LIN {X 0,Y 566.191,Z 469.084,A -85,B 0,C 180,E1 -2638.953,E2 -2638.953} C_VEL
LIN {X 0,Y 566.2,Z 469.079,A -85,B 0,C 180,E1 -2641.421,E2 -2641.421} C_VEL
LIN {X 0,Y 566.208,Z 469.076,A -85,B 0,C 180,E1 -2643.955,E2 -2643.955} C_VEL
LIN {X 0,Y 566.197,Z 469.068,A -85,B 0,C 180,E1 -2646.569,E2 -2646.569} C_VEL
LIN {X 0,Y 566.219,Z 469.081,A -85,B 0,C 180,E1 -2649.272,E2 -2649.272} C_VEL
LIN {X 0,Y 566.211,Z 469.073,A -85,B 0,C 180,E1 -2652.086,E2 -2652.086} C_VEL
LIN {X 0,Y 566.169,Z 469.084,A -85,B 0,C 180,E1 -2655.035,E2 -2655.035} C_VEL
LIN {X 0,Y 566.186,Z 469.078,A -85,B 0,C 180,E1 -2657.91,E2 -2657.91} C_VEL
LIN {X 0,Y 566.217,Z 469.076,A -85,B 0,C 180,E1 -2660.726,E2 -2660.726} C_VEL
LIN {X 0,Y 566.212,Z 469.077,A -85,B 0,C 180,E1 -2663.783,E2 -2663.783} C_VEL
LIN {X 0,Y 566.206,Z 469.073,A -85,B 0,C 180,E1 -2666.265,E2 -2666.265} C_VEL
LIN {X 0,Y 566.192,Z 469.08,A -85,B 0,C 180,E1 -2668.921,E2 -2668.921} C_VEL
LIN {X 0,Y 566.221,Z 469.073,A -85,B 0,C 180,E1 -2671.858,E2 -2671.858} C_VEL
LIN {X 0,Y 566.219,Z 469.073,A -85,B 0,C 180,E1 -2674.251,E2 -2674.251} C_VEL
LIN {X 0,Y 566.183,Z 469.079,A -85,B 0,C 180,E1 -2676.713,E2 -2676.713} C_VEL
LIN {X 0,Y 566.211,Z 469.078,A -85,B 0,C 180,E1 -2679.662,E2 -2679.662} C_VEL
LIN {X 0,Y 566.195,Z 469.077,A -85,B 0,C 180,E1 -2682.668,E2 -2682.668} C_VEL
LIN {X 0,Y 566.224,Z 469.075,A -85,B 0,C 180,E1 -2685.626,E2 -2685.626} C_VEL
LIN {X 0,Y 566.224,Z 469.072,A -85,B 0,C 180,E1 -2688.675,E2 -2688.675} C_VEL
LIN {X 0,Y 566.24,Z 469.081,A -85,B 0,C 180,E1 -2691.434,E2 -2691.434} C_VEL
LIN {X 0,Y 566.252,Z 469.065,A -85,B 0,C 180,E1 -2694.301,E2 -2694.301} C_VEL
LIN {X 0,Y 566.272,Z 469.071,A -85,B 0,C 180,E1 -2697.866,E2 -2697.866} C_VEL
LIN {X 0,Y 566.298,Z 469.062,A -85,B 0,C 180,E1 -2700.711,E2 -2700.711} C_VEL
LIN {X 0,Y 566.27,Z 469.064,A -85,B 0,C 180,E1 -2702.845,E2 -2702.845} C_VEL
LIN {X 0,Y 566.25,Z 469.077,A -85,B 0,C 180,E1 -2705.698,E2 -2705.698} C_VEL
LIN {X 0,Y 566.239,Z 469.069,A -85,B 0,C 180,E1 -2708.565,E2 -2708.565} C_VEL
LIN {X 0,Y 566.241,Z 469.076,A -85,B 0,C 180,E1 -2711.454,E2 -2711.454} C_VEL
LIN {X 0,Y 566.223,Z 469.073,A -85,B 0,C 180,E1 -2714.507,E2 -2714.507} C_VEL
LIN {X 0,Y 566.194,Z 469.08,A -85,B 0,C 180,E1 -2717.331,E2 -2717.331} C_VEL
LIN {X 0,Y 566.21,Z 469.075,A -85,B 0,C 180,E1 -2720.337,E2 -2720.337} C_VEL
LIN {X 0,Y 566.179,Z 469.084,A -85,B 0,C 180,E1 -2723.404,E2 -2723.404} C_VEL
LIN {X 0,Y 566.217,Z 469.082,A -85,B 0,C 180,E1 -2725.748,E2 -2725.748} C_VEL
LIN {X 0,Y 566.207,Z 469.078,A -85,B 0,C 180,E1 -2727.497,E2 -2727.497} C_VEL
LIN {X 0,Y 565.529,Z 469.163,A -85,B 0,C 180,E1 -2728.09,E2 -2728.09} C_VEL
LIN {X 0,Y 562.664,Z 469.517,A -85,B 0,C 180,E1 -2729.054,E2 -2729.054} C_VEL
LIN {X 0,Y 560.253,Z 469.821,A -85,B 0,C 180,E1 -2729.83,E2 -2729.83} C_VEL
LIN {X 0,Y 559.224,Z 469.943,A -85,B 0,C 180,E1 -2730.428,E2 -2730.428} C_VEL
LIN {X 0,Y 559.143,Z 469.952,A -85,B 0,C 180,E1 -2730.631,E2 -2730.631} C_VEL
LIN {X 0,Y 559.169,Z 469.96,A -85,B 0,C 180,E1 -2733.574,E2 -2733.574} C_VEL
LIN {X 0,Y 559.16,Z 469.952,A -85,B 0,C 180,E1 -2736.449,E2 -2736.449} C_VEL
LIN {X 0,Y 559.17,Z 469.952,A -85,B 0,C 180,E1 -2738.934,E2 -2738.934} C_VEL
LIN {X 0,Y 559.183,Z 469.959,A -85,B 0,C 180,E1 -2741.768,E2 -2741.768} C_VEL
LIN {X 0,Y 559.131,Z 469.955,A -85,B 0,C 180,E1 -2744.739,E2 -2744.739} C_VEL
LIN {X 0,Y 559.165,Z 469.946,A -85,B 0,C 180,E1 -2747.258,E2 -2747.258} C_VEL
LIN {X 0,Y 559.179,Z 469.955,A -85,B 0,C 180,E1 -2750.135,E2 -2750.135} C_VEL
LIN {X 0,Y 559.14,Z 469.951,A -85,B 0,C 180,E1 -2752.893,E2 -2752.893} C_VEL
LIN {X 0,Y 559.149,Z 469.96,A -85,B 0,C 180,E1 -2755.556,E2 -2755.556} C_VEL
LIN {X 0,Y 559.165,Z 469.958,A -85,B 0,C 180,E1 -2758.138,E2 -2758.138} C_VEL
LIN {X 0,Y 559.151,Z 469.955,A -85,B 0,C 180,E1 -2760.647,E2 -2760.647} C_VEL
LIN {X 0,Y 559.166,Z 469.954,A -85,B 0,C 180,E1 -2763.173,E2 -2763.173} C_VEL
LIN {X 0,Y 559.152,Z 469.959,A -85,B 0,C 180,E1 -2765.495,E2 -2765.495} C_VEL
LIN {X 0,Y 559.167,Z 469.954,A -85,B 0,C 180,E1 -2768.624,E2 -2768.624} C_VEL
LIN {X 0,Y 559.166,Z 469.953,A -85,B 0,C 180,E1 -2770.927,E2 -2770.927} C_VEL
LIN {X 0,Y 559.164,Z 469.962,A -85,B 0,C 180,E1 -2773.948,E2 -2773.948} C_VEL
LIN {X 0,Y 559.169,Z 469.959,A -85,B 0,C 180,E1 -2776.184,E2 -2776.184} C_VEL
LIN {X 0,Y 559.191,Z 469.951,A -85,B 0,C 180,E1 -2779.134,E2 -2779.134} C_VEL
LIN {X 0,Y 559.202,Z 469.957,A -85,B 0,C 180,E1 -2782.054,E2 -2782.054} C_VEL
LIN {X 0,Y 559.248,Z 469.943,A -85,B 0,C 180,E1 -2784.953,E2 -2784.953} C_VEL
LIN {X 0,Y 559.252,Z 469.951,A -85,B 0,C 180,E1 -2787.839,E2 -2787.839} C_VEL
LIN {X 0,Y 559.268,Z 469.942,A -85,B 0,C 180,E1 -2790.72,E2 -2790.72} C_VEL
LIN {X 0,Y 559.235,Z 469.945,A -85,B 0,C 180,E1 -2792.881,E2 -2792.881} C_VEL
LIN {X 0,Y 559.225,Z 469.952,A -85,B 0,C 180,E1 -2795.77,E2 -2795.77} C_VEL
LIN {X 0,Y 559.183,Z 469.952,A -85,B 0,C 180,E1 -2798.674,E2 -2798.674} C_VEL
LIN {X 0,Y 559.202,Z 469.952,A -85,B 0,C 180,E1 -2801.6,E2 -2801.6} C_VEL
LIN {X 0,Y 559.196,Z 469.952,A -85,B 0,C 180,E1 -2804.595,E2 -2804.595} C_VEL
LIN {X 0,Y 559.159,Z 469.956,A -85,B 0,C 180,E1 -2807.556,E2 -2807.556} C_VEL
LIN {X 0,Y 559.168,Z 469.959,A -85,B 0,C 180,E1 -2809.837,E2 -2809.837} C_VEL
LIN {X 0,Y 559.137,Z 469.966,A -85,B 0,C 180,E1 -2812.152,E2 -2812.152} C_VEL
LIN {X 0,Y 559.174,Z 469.952,A -85,B 0,C 180,E1 -2815.187,E2 -2815.187} C_VEL
LIN {X 0,Y 559.186,Z 469.954,A -85,B 0,C 180,E1 -2817.711,E2 -2817.711} C_VEL
LIN {X 0,Y 559.163,Z 469.963,A -85,B 0,C 180,E1 -2820.181,E2 -2820.181} C_VEL
LIN {X 0,Y 559.169,Z 469.955,A -85,B 0,C 180,E1 -2822.714,E2 -2822.714} C_VEL
LIN {X 0,Y 559.15,Z 469.954,A -85,B 0,C 180,E1 -2825.322,E2 -2825.322} C_VEL
LIN {X 0,Y 559.129,Z 469.96,A -85,B 0,C 180,E1 -2828.017,E2 -2828.017} C_VEL
LIN {X 0,Y 559.169,Z 469.952,A -85,B 0,C 180,E1 -2830.81,E2 -2830.81} C_VEL
LIN {X 0,Y 559.156,Z 469.947,A -85,B 0,C 180,E1 -2833.731,E2 -2833.731} C_VEL
LIN {X 0,Y 559.159,Z 469.956,A -85,B 0,C 180,E1 -2836.801,E2 -2836.801} C_VEL
LIN {X 0,Y 559.167,Z 469.95,A -85,B 0,C 180,E1 -2839.189,E2 -2839.189} C_VEL
LIN {X 0,Y 559.126,Z 469.963,A -85,B 0,C 180,E1 -2841.982,E2 -2841.982} C_VEL
LIN {X 0,Y 559.152,Z 469.956,A -85,B 0,C 180,E1 -2844.782,E2 -2844.782} C_VEL
LIN {X 0,Y 559.165,Z 469.952,A -85,B 0,C 180,E1 -2847.361,E2 -2847.361} C_VEL
LIN {X 0,Y 559.18,Z 469.954,A -85,B 0,C 180,E1 -2850.135,E2 -2850.135} C_VEL
LIN {X 0,Y 559.173,Z 469.951,A -85,B 0,C 180,E1 -2853.17,E2 -2853.17} C_VEL
LIN {X 0,Y 559.147,Z 469.951,A -85,B 0,C 180,E1 -2855.495,E2 -2855.495} C_VEL
LIN {X 0,Y 559.167,Z 469.958,A -85,B 0,C 180,E1 -2858.624,E2 -2858.624} C_VEL
LIN {X 0,Y 559.162,Z 469.953,A -85,B 0,C 180,E1 -2860.926,E2 -2860.926} C_VEL
LIN {X 0,Y 559.161,Z 469.953,A -85,B 0,C 180,E1 -2863.948,E2 -2863.948} C_VEL
LIN {X 0,Y 559.164,Z 469.958,A -85,B 0,C 180,E1 -2866.184,E2 -2866.184} C_VEL
LIN {X 0,Y 559.201,Z 469.945,A -85,B 0,C 180,E1 -2869.134,E2 -2869.134} C_VEL
LIN {X 0,Y 559.201,Z 469.949,A -85,B 0,C 180,E1 -2872.054,E2 -2872.054} C_VEL
LIN {X 0,Y 559.251,Z 469.943,A -85,B 0,C 180,E1 -2874.954,E2 -2874.954} C_VEL
LIN {X 0,Y 559.243,Z 469.939,A -85,B 0,C 180,E1 -2877.84,E2 -2877.84} C_VEL
LIN {X 0,Y 559.268,Z 469.945,A -85,B 0,C 180,E1 -2880.72,E2 -2880.72} C_VEL
LIN {X 0,Y 559.236,Z 469.946,A -85,B 0,C 180,E1 -2882.882,E2 -2882.882} C_VEL
LIN {X 0,Y 559.221,Z 469.94,A -85,B 0,C 180,E1 -2885.771,E2 -2885.771} C_VEL
LIN {X 0,Y 559.194,Z 469.957,A -85,B 0,C 180,E1 -2888.675,E2 -2888.675} C_VEL
LIN {X 0,Y 559.196,Z 469.947,A -85,B 0,C 180,E1 -2891.601,E2 -2891.601} C_VEL
LIN {X 0,Y 559.19,Z 469.955,A -85,B 0,C 180,E1 -2894.596,E2 -2894.596} C_VEL
LIN {X 0,Y 559.155,Z 469.953,A -85,B 0,C 180,E1 -2897.557,E2 -2897.557} C_VEL
LIN {X 0,Y 559.166,Z 469.95,A -85,B 0,C 180,E1 -2899.838,E2 -2899.838} C_VEL
LIN {X 0,Y 559.135,Z 469.957,A -85,B 0,C 180,E1 -2902.153,E2 -2902.153} C_VEL
LIN {X 0,Y 559.172,Z 469.952,A -85,B 0,C 180,E1 -2905.188,E2 -2905.188} C_VEL
LIN {X 0,Y 559.188,Z 469.946,A -85,B 0,C 180,E1 -2907.712,E2 -2907.712} C_VEL
LIN {X 0,Y 559.156,Z 469.957,A -85,B 0,C 180,E1 -2911.02,E2 -2911.02} C_VEL
LIN {X 0,Y 559.162,Z 469.951,A -85,B 0,C 180,E1 -2913.95,E2 -2913.95} C_VEL
LIN {X 0,Y 559.163,Z 469.959,A -85,B 0,C 180,E1 -2916.449,E2 -2916.449} C_VEL
LIN {X 0,Y 559.173,Z 469.958,A -85,B 0,C 180,E1 -2918.934,E2 -2918.934} C_VEL
LIN {X 0,Y 559.164,Z 469.951,A -85,B 0,C 180,E1 -2921.77,E2 -2921.77} C_VEL
LIN {X 0,Y 559.135,Z 469.965,A -85,B 0,C 180,E1 -2924.74,E2 -2924.74} C_VEL
LIN {X 0,Y 559.161,Z 469.954,A -85,B 0,C 180,E1 -2927.258,E2 -2927.258} C_VEL
LIN {X 0,Y 559.182,Z 469.952,A -85,B 0,C 180,E1 -2930.136,E2 -2930.136} C_VEL
LIN {X 0,Y 559.138,Z 469.95,A -85,B 0,C 180,E1 -2932.892,E2 -2932.892} C_VEL
LIN {X 0,Y 559.164,Z 469.954,A -85,B 0,C 180,E1 -2936.052,E2 -2936.052} C_VEL
LIN {X 0,Y 559.162,Z 469.951,A -85,B 0,C 180,E1 -2938.982,E2 -2938.982} C_VEL
LIN {X 0,Y 559.168,Z 469.953,A -85,B 0,C 180,E1 -2941.619,E2 -2941.619} C_VEL
LIN {X 0,Y 559.2,Z 470.086,A -85,B 0,C 180,E1 -2943.503,E2 -2943.503} C_VEL
LIN {X 0,Y 560.282,Z 475.94,A -85,B 0,C 180,E1 -2944.575,E2 -2944.575} C_VEL
LIN {X 0,Y 560.031,Z 493.496,A -85,B 0,C 180,E1 -2947.496,E2 -2947.496} C_VEL
LIN {X 0,Y 559.744,Z 510.701,A -85,B 0,C 180,E1 -2950.336,E2 -2950.336} C_VEL
LIN {X 0,Y 559.551,Z 526.039,A -85,B 0,C 180,E1 -2952.795,E2 -2952.795} C_VEL
LIN {X 0,Y 560.706,Z 532.012,A -85,B 0,C 180,E1 -2952.937,E2 -2952.937} C_VEL
LIN {X 0,Y 561.014,Z 537.106,A -85,B 0,C 180,E1 -2953.014,E2 -2953.014} C_VEL
LIN {X 0,Y 560.621,Z 661.281,A -85,B 0,C 180,E1 -2954.644,E2 -2954.644} C_VEL
LIN {X 0,Y 560.468,Z 673.415,A -85,B 0,C 180,E1 -2954.905,E2 -2954.905} C_VEL
LIN {X 0,Y 560.366,Z 685.467,A -85,B 0,C 180,E1 -2955.275,E2 -2955.275} C_VEL
LIN {X 0,Y 560.152,Z 699.181,A -85,B 0,C 180,E1 -2955.839,E2 -2955.839} C_VEL
LIN {X 0,Y 559.865,Z 712.711,A -85,B 0,C 180,E1 -2956.572,E2 -2956.572} C_VEL
LIN {X 0,Y 559.702,Z 723.64,A -85,B 0,C 180,E1 -2957.306,E2 -2957.306} C_VEL
LIN {X 0,Y 559.514,Z 733.886,A -85,B 0,C 180,E1 -2958.131,E2 -2958.131} C_VEL
LIN {X 0,Y 559.35,Z 744.375,A -85,B 0,C 180,E1 -2959.137,E2 -2959.137} C_VEL
LIN {X 0,Y 559.143,Z 753.825,A -85,B 0,C 180,E1 -2960.231,E2 -2960.231} C_VEL
LIN {X 0,Y 559.053,Z 761.624,A -85,B 0,C 180,E1 -2961.324,E2 -2961.324} C_VEL
LIN {X 0,Y 558.966,Z 768.13,A -85,B 0,C 180,E1 -2962.414,E2 -2962.414} C_VEL
LIN {X 0,Y 558.872,Z 773.519,A -85,B 0,C 180,E1 -2963.502,E2 -2963.502} C_VEL
LIN {X 0,Y 558.858,Z 777.921,A -85,B 0,C 180,E1 -2964.588,E2 -2964.588} C_VEL
LIN {X 0,Y 558.865,Z 781.441,A -85,B 0,C 180,E1 -2965.673,E2 -2965.673} C_VEL
LIN {X 0,Y 558.825,Z 783.323,A -85,B 0,C 180,E1 -2966.395,E2 -2966.395} C_VEL
LIN {X 0,Y 558.743,Z 786.005,A -85,B 0,C 180,E1 -2967.837,E2 -2967.837} C_VEL
LIN {X 0,Y 558.738,Z 787.29,A -85,B 0,C 180,E1 -2969.279,E2 -2969.279} C_VEL
LIN {X 0,Y 558.738,Z 787.5,A -85,B 0,C 180,E1 -2970,E2 -2970} C_VEL
LIN {X 0,Y 558.74,Z 786.808,A -85,B 0,C 180,E1 -2971.441,E2 -2971.441} C_VEL
LIN {X 0,Y 558.743,Z 786.005,A -85,B 0,C 180,E1 -2972.163,E2 -2972.163} C_VEL
LIN {X 0,Y 558.825,Z 783.323,A -85,B 0,C 180,E1 -2973.605,E2 -2973.605} C_VEL
LIN {X 0,Y 558.82,Z 780.397,A -85,B 0,C 180,E1 -2974.689,E2 -2974.689} C_VEL
LIN {X 0,Y 558.882,Z 775.086,A -85,B 0,C 180,E1 -2976.136,E2 -2976.136} C_VEL
LIN {X 0,Y 558.907,Z 770.03,A -85,B 0,C 180,E1 -2977.224,E2 -2977.224} C_VEL
LIN {X 0,Y 559.006,Z 763.885,A -85,B 0,C 180,E1 -2978.313,E2 -2978.313} C_VEL
LIN {X 0,Y 559.117,Z 756.524,A -85,B 0,C 180,E1 -2979.405,E2 -2979.405} C_VEL
LIN {X 0,Y 559.267,Z 747.714,A -85,B 0,C 180,E1 -2980.498,E2 -2980.498} C_VEL
LIN {X 0,Y 559.454,Z 737.023,A -85,B 0,C 180,E1 -2981.595,E2 -2981.595} C_VEL
LIN {X 0,Y 559.637,Z 726.113,A -85,B 0,C 180,E1 -2982.511,E2 -2982.511} C_VEL
LIN {X 0,Y 559.827,Z 715.633,A -85,B 0,C 180,E1 -2983.244,E2 -2983.244} C_VEL
LIN {X 0,Y 560.047,Z 704.551,A -85,B 0,C 180,E1 -2983.886,E2 -2983.886} C_VEL
LIN {X 0,Y 560.232,Z 692.882,A -85,B 0,C 180,E1 -2984.437,E2 -2984.437} C_VEL
LIN {X 0,Y 560.411,Z 679.335,A -85,B 0,C 180,E1 -2984.933,E2 -2984.933} C_VEL
LIN {X 0,Y 560.563,Z 663.998,A -85,B 0,C 180,E1 -2985.311,E2 -2985.311} C_VEL
LIN {X 0,Y 560.693,Z 637.754,A -85,B 0,C 180,E1 -2985.68,E2 -2985.68} C_VEL
LIN {X 0,Y 560.863,Z 532.996,A -85,B 0,C 180,E1 -2987.045,E2 -2987.045} C_VEL
LIN {X 0,Y 559.547,Z 526.183,A -85,B 0,C 180,E1 -2987.195,E2 -2987.195} C_VEL
LIN {X 0,Y 559.567,Z 522.568,A -85,B 0,C 180,E1 -2987.732,E2 -2987.732} C_VEL
LIN {X 0,Y 559.837,Z 503.962,A -85,B 0,C 180,E1 -2990.771,E2 -2990.771} C_VEL
LIN {X 0,Y 560.096,Z 488.81,A -85,B 0,C 180,E1 -2993.281,E2 -2993.281} C_VEL
LIN {X 0,Y 560.269,Z 475.96,A -85,B 0,C 180,E1 -2995.422,E2 -2995.422} C_VEL
LIN {X 0,Y 559.19,Z 470.039,A -85,B 0,C 180,E1 -2996.518,E2 -2996.518} C_VEL
LIN {X 0,Y 559.142,Z 469.962,A -85,B 0,C 180,E1 -2999.353,E2 -2999.353} C_VEL
LIN {X 0,Y 559.169,Z 469.952,A -85,B 0,C 180,E1 -3001.862,E2 -3001.862} C_VEL
LIN {X 0,Y 559.141,Z 469.957,A -85,B 0,C 180,E1 -3004.444,E2 -3004.444} C_VEL
LIN {X 0,Y 559.138,Z 469.95,A -85,B 0,C 180,E1 -3007.108,E2 -3007.108} C_VEL
LIN {X 0,Y 559.166,Z 469.953,A -85,B 0,C 180,E1 -3009.942,E2 -3009.942} C_VEL
LIN {X 0,Y 559.161,Z 469.954,A -85,B 0,C 180,E1 -3012.742,E2 -3012.742} C_VEL
LIN {X 0,Y 559.148,Z 469.957,A -85,B 0,C 180,E1 -3015.76,E2 -3015.76} C_VEL
LIN {X 0,Y 559.164,Z 469.951,A -85,B 0,C 180,E1 -3018.23,E2 -3018.23} C_VEL
LIN {X 0,Y 559.172,Z 469.96,A -85,B 0,C 180,E1 -3021.19,E2 -3021.19} C_VEL
LIN {X 0,Y 559.167,Z 469.955,A -85,B 0,C 180,E1 -3023.791,E2 -3023.791} C_VEL
LIN {X 0,Y 559.159,Z 469.951,A -85,B 0,C 180,E1 -3026.425,E2 -3026.425} C_VEL
LIN {X 0,Y 559.156,Z 469.957,A -85,B 0,C 180,E1 -3028.98,E2 -3028.98} C_VEL
LIN {X 0,Y 559.188,Z 469.946,A -85,B 0,C 180,E1 -3032.288,E2 -3032.288} C_VEL
LIN {X 0,Y 559.172,Z 469.952,A -85,B 0,C 180,E1 -3034.812,E2 -3034.812} C_VEL
LIN {X 0,Y 559.135,Z 469.957,A -85,B 0,C 180,E1 -3037.847,E2 -3037.847} C_VEL
LIN {X 0,Y 559.19,Z 469.947,A -85,B 0,C 180,E1 -3040.491,E2 -3040.491} C_VEL
LIN {X 0,Y 559.176,Z 469.957,A -85,B 0,C 180,E1 -3043.197,E2 -3043.197} C_VEL
LIN {X 0,Y 559.164,Z 469.948,A -85,B 0,C 180,E1 -3046.184,E2 -3046.184} C_VEL
LIN {X 0,Y 559.187,Z 469.953,A -85,B 0,C 180,E1 -3049.133,E2 -3049.133} C_VEL
LIN {X 0,Y 559.2,Z 469.948,A -85,B 0,C 180,E1 -3052.053,E2 -3052.053} C_VEL
LIN {X 0,Y 559.25,Z 469.939,A -85,B 0,C 180,E1 -3054.953,E2 -3054.953} C_VEL
LIN {X 0,Y 559.243,Z 469.947,A -85,B 0,C 180,E1 -3057.839,E2 -3057.839} C_VEL
LIN {X 0,Y 559.268,Z 469.937,A -85,B 0,C 180,E1 -3060.72,E2 -3060.72} C_VEL
LIN {X 0,Y 559.236,Z 469.94,A -85,B 0,C 180,E1 -3062.881,E2 -3062.881} C_VEL
LIN {X 0,Y 559.22,Z 469.951,A -85,B 0,C 180,E1 -3065.77,E2 -3065.77} C_VEL
LIN {X 0,Y 559.194,Z 469.946,A -85,B 0,C 180,E1 -3068.674,E2 -3068.674} C_VEL
LIN {X 0,Y 559.199,Z 469.955,A -85,B 0,C 180,E1 -3071.6,E2 -3071.6} C_VEL
LIN {X 0,Y 559.188,Z 469.949,A -85,B 0,C 180,E1 -3074.595,E2 -3074.595} C_VEL
LIN {X 0,Y 559.154,Z 469.959,A -85,B 0,C 180,E1 -3077.557,E2 -3077.557} C_VEL
LIN {X 0,Y 559.165,Z 469.959,A -85,B 0,C 180,E1 -3079.837,E2 -3079.837} C_VEL
LIN {X 0,Y 559.132,Z 469.958,A -85,B 0,C 180,E1 -3082.153,E2 -3082.153} C_VEL
LIN {X 0,Y 559.169,Z 469.951,A -85,B 0,C 180,E1 -3085.187,E2 -3085.187} C_VEL
LIN {X 0,Y 559.185,Z 469.959,A -85,B 0,C 180,E1 -3087.711,E2 -3087.711} C_VEL
LIN {X 0,Y 559.143,Z 469.952,A -85,B 0,C 180,E1 -3090.631,E2 -3090.631} C_VEL
LIN {X 0,Y 558.48,Z 470.039,A -85,B 0,C 180,E1 -3091.233,E2 -3091.233} C_VEL
LIN {X 0,Y 555.617,Z 470.396,A -85,B 0,C 180,E1 -3092.209,E2 -3092.209} C_VEL
LIN {X 0,Y 553.206,Z 470.696,A -85,B 0,C 180,E1 -3092.994,E2 -3092.994} C_VEL
LIN {X 0,Y 552.188,Z 470.83,A -85,B 0,C 180,E1 -3093.601,E2 -3093.601} C_VEL
LIN {X 0,Y 552.115,Z 470.832,A -85,B 0,C 180,E1 -3093.806,E2 -3093.806} C_VEL
LIN {X 0,Y 552.103,Z 470.83,A -85,B 0,C 180,E1 -3096.747,E2 -3096.747} C_VEL
LIN {X 0,Y 552.126,Z 470.836,A -85,B 0,C 180,E1 -3099.527,E2 -3099.527} C_VEL
LIN {X 0,Y 552.122,Z 470.831,A -85,B 0,C 180,E1 -3102.426,E2 -3102.426} C_VEL
LIN {X 0,Y 552.092,Z 470.839,A -85,B 0,C 180,E1 -3105.563,E2 -3105.563} C_VEL
LIN {X 0,Y 552.164,Z 470.823,A -85,B 0,C 180,E1 -3108.673,E2 -3108.673} C_VEL
LIN {X 0,Y 552.114,Z 470.835,A -85,B 0,C 180,E1 -3111.412,E2 -3111.412} C_VEL
LIN {X 0,Y 552.106,Z 470.836,A -85,B 0,C 180,E1 -3114.159,E2 -3114.159} C_VEL
LIN {X 0,Y 552.117,Z 470.831,A -85,B 0,C 180,E1 -3116.815,E2 -3116.815} C_VEL
LIN {X 0,Y 552.108,Z 470.835,A -85,B 0,C 180,E1 -3119.392,E2 -3119.392} C_VEL
LIN {X 0,Y 552.12,Z 470.84,A -85,B 0,C 180,E1 -3121.903,E2 -3121.903} C_VEL
LIN {X 0,Y 552.15,Z 470.828,A -85,B 0,C 180,E1 -3124.65,E2 -3124.65} C_VEL
LIN {X 0,Y 552.091,Z 470.839,A -85,B 0,C 180,E1 -3127.55,E2 -3127.55} C_VEL
LIN {X 0,Y 552.152,Z 470.828,A -85,B 0,C 180,E1 -3130.675,E2 -3130.675} C_VEL
LIN {X 0,Y 552.114,Z 470.839,A -85,B 0,C 180,E1 -3133.738,E2 -3133.738} C_VEL
LIN {X 0,Y 552.132,Z 470.838,A -85,B 0,C 180,E1 -3136.005,E2 -3136.005} C_VEL
LIN {X 0,Y 552.159,Z 470.826,A -85,B 0,C 180,E1 -3138.994,E2 -3138.994} C_VEL
LIN {X 0,Y 552.156,Z 470.835,A -85,B 0,C 180,E1 -3141.952,E2 -3141.952} C_VEL
LIN {X 0,Y 552.223,Z 470.819,A -85,B 0,C 180,E1 -3144.889,E2 -3144.889} C_VEL
LIN {X 0,Y 552.223,Z 470.826,A -85,B 0,C 180,E1 -3147.812,E2 -3147.812} C_VEL
LIN {X 0,Y 552.238,Z 470.818,A -85,B 0,C 180,E1 -3150.729,E2 -3150.729} C_VEL
LIN {X 0,Y 552.202,Z 470.821,A -85,B 0,C 180,E1 -3152.918,E2 -3152.918} C_VEL
LIN {X 0,Y 552.196,Z 470.829,A -85,B 0,C 180,E1 -3155.844,E2 -3155.844} C_VEL
LIN {X 0,Y 552.154,Z 470.827,A -85,B 0,C 180,E1 -3158.786,E2 -3158.786} C_VEL
LIN {X 0,Y 552.159,Z 470.831,A -85,B 0,C 180,E1 -3161.75,E2 -3161.75} C_VEL
LIN {X 0,Y 552.133,Z 470.831,A -85,B 0,C 180,E1 -3164.748,E2 -3164.748} C_VEL
LIN {X 0,Y 552.11,Z 470.838,A -85,B 0,C 180,E1 -3167.788,E2 -3167.788} C_VEL
LIN {X 0,Y 552.126,Z 470.839,A -85,B 0,C 180,E1 -3170.101,E2 -3170.101} C_VEL
LIN {X 0,Y 552.091,Z 470.839,A -85,B 0,C 180,E1 -3172.45,E2 -3172.45} C_VEL
LIN {X 0,Y 552.15,Z 470.828,A -85,B 0,C 180,E1 -3175.35,E2 -3175.35} C_VEL
LIN {X 0,Y 552.12,Z 470.84,A -85,B 0,C 180,E1 -3178.097,E2 -3178.097} C_VEL
LIN {X 0,Y 552.108,Z 470.835,A -85,B 0,C 180,E1 -3180.608,E2 -3180.608} C_VEL
LIN {X 0,Y 552.117,Z 470.831,A -85,B 0,C 180,E1 -3183.185,E2 -3183.185} C_VEL
LIN {X 0,Y 552.106,Z 470.836,A -85,B 0,C 180,E1 -3185.841,E2 -3185.841} C_VEL
LIN {X 0,Y 552.119,Z 470.831,A -85,B 0,C 180,E1 -3189.062,E2 -3189.062} C_VEL
LIN {X 0,Y 552.134,Z 470.827,A -85,B 0,C 180,E1 -3191.443,E2 -3191.443} C_VEL
LIN {X 0,Y 552.089,Z 470.838,A -85,B 0,C 180,E1 -3194.532,E2 -3194.532} C_VEL
LIN {X 0,Y 552.122,Z 470.831,A -85,B 0,C 180,E1 -3197.584,E2 -3197.584} C_VEL
LIN {X 0,Y 552.126,Z 470.836,A -85,B 0,C 180,E1 -3200.473,E2 -3200.473} C_VEL
LIN {X 0,Y 552.105,Z 470.83,A -85,B 0,C 180,E1 -3203.315,E2 -3203.315} C_VEL
LIN {X 0,Y 552.131,Z 470.832,A -85,B 0,C 180,E1 -3205.94,E2 -3205.94} C_VEL
LIN {X 0,Y 552.108,Z 470.834,A -85,B 0,C 180,E1 -3208.54,E2 -3208.54} C_VEL
LIN {X 0,Y 552.117,Z 470.83,A -85,B 0,C 180,E1 -3211.437,E2 -3211.437} C_VEL
LIN {X 0,Y 552.128,Z 470.835,A -85,B 0,C 180,E1 -3214.356,E2 -3214.356} C_VEL
LIN {X 0,Y 552.1,Z 470.835,A -85,B 0,C 180,E1 -3216.758,E2 -3216.758} C_VEL
LIN {X 0,Y 552.116,Z 470.831,A -85,B 0,C 180,E1 -3219.12,E2 -3219.12} C_VEL
LIN {X 0,Y 552.122,Z 470.827,A -85,B 0,C 180,E1 -3221.445,E2 -3221.445} C_VEL
LIN {X 0,Y 552.111,Z 470.829,A -85,B 0,C 180,E1 -3223.738,E2 -3223.738} C_VEL
LIN {X 0,Y 552.126,Z 470.832,A -85,B 0,C 180,E1 -3226.005,E2 -3226.005} C_VEL
LIN {X 0,Y 552.168,Z 470.822,A -85,B 0,C 180,E1 -3228.994,E2 -3228.994} C_VEL
LIN {X 0,Y 552.155,Z 470.825,A -85,B 0,C 180,E1 -3231.952,E2 -3231.952} C_VEL
LIN {X 0,Y 552.225,Z 470.819,A -85,B 0,C 180,E1 -3234.889,E2 -3234.889} C_VEL
LIN {X 0,Y 552.215,Z 470.814,A -85,B 0,C 180,E1 -3237.812,E2 -3237.812} C_VEL
LIN {X 0,Y 552.237,Z 470.821,A -85,B 0,C 180,E1 -3240.73,E2 -3240.73} C_VEL
LIN {X 0,Y 552.202,Z 470.822,A -85,B 0,C 180,E1 -3242.918,E2 -3242.918} C_VEL
LIN {X 0,Y 552.191,Z 470.816,A -85,B 0,C 180,E1 -3245.844,E2 -3245.844} C_VEL
LIN {X 0,Y 552.162,Z 470.831,A -85,B 0,C 180,E1 -3248.786,E2 -3248.786} C_VEL
LIN {X 0,Y 552.153,Z 470.825,A -85,B 0,C 180,E1 -3251.751,E2 -3251.751} C_VEL
LIN {X 0,Y 552.128,Z 470.835,A -85,B 0,C 180,E1 -3254.749,E2 -3254.749} C_VEL
LIN {X 0,Y 552.107,Z 470.832,A -85,B 0,C 180,E1 -3257.789,E2 -3257.789} C_VEL
LIN {X 0,Y 552.126,Z 470.829,A -85,B 0,C 180,E1 -3260.102,E2 -3260.102} C_VEL
LIN {X 0,Y 552.088,Z 470.838,A -85,B 0,C 180,E1 -3262.451,E2 -3262.451} C_VEL
LIN {X 0,Y 552.149,Z 470.826,A -85,B 0,C 180,E1 -3265.352,E2 -3265.352} C_VEL
LIN {X 0,Y 552.12,Z 470.829,A -85,B 0,C 180,E1 -3268.098,E2 -3268.098} C_VEL
LIN {X 0,Y 552.101,Z 470.842,A -85,B 0,C 180,E1 -3270.61,E2 -3270.61} C_VEL
LIN {X 0,Y 552.117,Z 470.831,A -85,B 0,C 180,E1 -3273.186,E2 -3273.186} C_VEL
LIN {X 0,Y 552.108,Z 470.832,A -85,B 0,C 180,E1 -3275.842,E2 -3275.842} C_VEL
LIN {X 0,Y 552.12,Z 470.835,A -85,B 0,C 180,E1 -3279.063,E2 -3279.063} C_VEL
LIN {X 0,Y 552.125,Z 470.829,A -85,B 0,C 180,E1 -3281.446,E2 -3281.446} C_VEL
LIN {X 0,Y 552.091,Z 470.841,A -85,B 0,C 180,E1 -3284.533,E2 -3284.533} C_VEL
LIN {X 0,Y 552.128,Z 470.827,A -85,B 0,C 180,E1 -3287.585,E2 -3287.585} C_VEL
LIN {X 0,Y 552.131,Z 470.834,A -85,B 0,C 180,E1 -3290.474,E2 -3290.474} C_VEL
LIN {X 0,Y 552.104,Z 470.821,A -85,B 0,C 180,E1 -3293.318,E2 -3293.318} C_VEL
LIN {X 0,Y 552.125,Z 470.831,A -85,B 0,C 180,E1 -3295.94,E2 -3295.94} C_VEL
LIN {X 0,Y 552.118,Z 470.831,A -85,B 0,C 180,E1 -3298.541,E2 -3298.541} C_VEL
LIN {X 0,Y 552.124,Z 470.831,A -85,B 0,C 180,E1 -3301.439,E2 -3301.439} C_VEL
LIN {X 0,Y 552.17,Z 471.047,A -85,B 0,C 180,E1 -3303.339,E2 -3303.339} C_VEL
LIN {X 0,Y 553.38,Z 477.467,A -85,B 0,C 180,E1 -3304.524,E2 -3304.524} C_VEL
LIN {X 0,Y 553.086,Z 495.719,A -85,B 0,C 180,E1 -3307.592,E2 -3307.592} C_VEL
LIN {X 0,Y 552.742,Z 512.913,A -85,B 0,C 180,E1 -3310.445,E2 -3310.445} C_VEL
LIN {X 0,Y 552.607,Z 526.043,A -85,B 0,C 180,E1 -3312.572,E2 -3312.572} C_VEL
LIN {X 0,Y 553.554,Z 531.047,A -85,B 0,C 180,E1 -3312.697,E2 -3312.697} C_VEL
LIN {X 0,Y 554.245,Z 535.775,A -85,B 0,C 180,E1 -3312.782,E2 -3312.782} C_VEL
LIN {X 0,Y 553.785,Z 661.233,A -85,B 0,C 180,E1 -3314.449,E2 -3314.449} C_VEL
LIN {X 0,Y 553.635,Z 672.798,A -85,B 0,C 180,E1 -3314.699,E2 -3314.699} C_VEL
LIN {X 0,Y 553.503,Z 683.85,A -85,B 0,C 180,E1 -3315.033,E2 -3315.033} C_VEL
LIN {X 0,Y 553.3,Z 696.078,A -85,B 0,C 180,E1 -3315.519,E2 -3315.519} C_VEL
LIN {X 0,Y 553.025,Z 709.692,A -85,B 0,C 180,E1 -3316.215,E2 -3316.215} C_VEL
LIN {X 0,Y 552.771,Z 722.391,A -85,B 0,C 180,E1 -3317.051,E2 -3317.051} C_VEL
LIN {X 0,Y 552.531,Z 732.822,A -85,B 0,C 180,E1 -3317.885,E2 -3317.885} C_VEL
LIN {X 0,Y 552.394,Z 741.995,A -85,B 0,C 180,E1 -3318.754,E2 -3318.754} C_VEL
LIN {X 0,Y 552.178,Z 750.814,A -85,B 0,C 180,E1 -3319.736,E2 -3319.736} C_VEL
LIN {X 0,Y 552.04,Z 759.177,A -85,B 0,C 180,E1 -3320.843,E2 -3320.843} C_VEL
LIN {X 0,Y 551.913,Z 767.145,A -85,B 0,C 180,E1 -3322.132,E2 -3322.132} C_VEL
LIN {X 0,Y 551.822,Z 773.512,A -85,B 0,C 180,E1 -3323.418,E2 -3323.418} C_VEL
LIN {X 0,Y 551.791,Z 777.915,A -85,B 0,C 180,E1 -3324.519,E2 -3324.519} C_VEL
LIN {X 0,Y 551.759,Z 781.434,A -85,B 0,C 180,E1 -3325.617,E2 -3325.617} C_VEL
LIN {X 0,Y 551.74,Z 783.324,A -85,B 0,C 180,E1 -3326.348,E2 -3326.348} C_VEL
LIN {X 0,Y 551.654,Z 786.001,A -85,B 0,C 180,E1 -3327.81,E2 -3327.81} C_VEL
LIN {X 0,Y 551.638,Z 787.283,A -85,B 0,C 180,E1 -3329.27,E2 -3329.27} C_VEL
LIN {X 0,Y 551.639,Z 787.5,A -85,B 0,C 180,E1 -3330,E2 -3330} C_VEL
LIN {X 0,Y 551.639,Z 786.805,A -85,B 0,C 180,E1 -3331.46,E2 -3331.46} C_VEL
LIN {X 0,Y 551.654,Z 786.001,A -85,B 0,C 180,E1 -3332.19,E2 -3332.19} C_VEL
LIN {X 0,Y 551.74,Z 783.324,A -85,B 0,C 180,E1 -3333.652,E2 -3333.652} C_VEL
LIN {X 0,Y 551.716,Z 779.17,A -85,B 0,C 180,E1 -3335.116,E2 -3335.116} C_VEL
LIN {X 0,Y 551.782,Z 774.594,A -85,B 0,C 180,E1 -3336.329,E2 -3336.329} C_VEL
LIN {X 0,Y 551.833,Z 770.022,A -85,B 0,C 180,E1 -3337.317,E2 -3337.317} C_VEL
LIN {X 0,Y 551.961,Z 763.879,A -85,B 0,C 180,E1 -3338.42,E2 -3338.42} C_VEL
LIN {X 0,Y 552.068,Z 756.516,A -85,B 0,C 180,E1 -3339.526,E2 -3339.526} C_VEL
LIN {X 0,Y 552.237,Z 747.704,A -85,B 0,C 180,E1 -3340.634,E2 -3340.634} C_VEL
LIN {X 0,Y 552.464,Z 737.025,A -85,B 0,C 180,E1 -3341.744,E2 -3341.744} C_VEL
LIN {X 0,Y 552.667,Z 726.101,A -85,B 0,C 180,E1 -3342.671,E2 -3342.671} C_VEL
LIN {X 0,Y 552.863,Z 715.619,A -85,B 0,C 180,E1 -3343.414,E2 -3343.414} C_VEL
LIN {X 0,Y 553.14,Z 704.54,A -85,B 0,C 180,E1 -3344.063,E2 -3344.063} C_VEL
LIN {X 0,Y 553.351,Z 692.862,A -85,B 0,C 180,E1 -3344.621,E2 -3344.621} C_VEL
LIN {X 0,Y 553.544,Z 679.573,A -85,B 0,C 180,E1 -3345.114,E2 -3345.114} C_VEL
LIN {X 0,Y 553.729,Z 663.95,A -85,B 0,C 180,E1 -3345.505,E2 -3345.505} C_VEL
LIN {X 0,Y 553.869,Z 639.543,A -85,B 0,C 180,E1 -3345.855,E2 -3345.855} C_VEL
LIN {X 0,Y 554.144,Z 534.259,A -85,B 0,C 180,E1 -3347.241,E2 -3347.241} C_VEL
LIN {X 0,Y 552.586,Z 526.242,A -85,B 0,C 180,E1 -3347.416,E2 -3347.416} C_VEL
LIN {X 0,Y 552.603,Z 522.568,A -85,B 0,C 180,E1 -3347.963,E2 -3347.963} C_VEL
LIN {X 0,Y 552.975,Z 502.784,A -85,B 0,C 180,E1 -3351.236,E2 -3351.236} C_VEL
LIN {X 0,Y 553.25,Z 485.111,A -85,B 0,C 180,E1 -3354.184,E2 -3354.184} C_VEL
LIN {X 0,Y 553.267,Z 476.842,A -85,B 0,C 180,E1 -3355.592,E2 -3355.592} C_VEL
LIN {X 0,Y 552.138,Z 470.915,A -85,B 0,C 180,E1 -3356.704,E2 -3356.704} C_VEL
LIN {X 0,Y 552.112,Z 470.832,A -85,B 0,C 180,E1 -3359.764,E2 -3359.764} C_VEL
LIN {X 0,Y 552.117,Z 470.829,A -85,B 0,C 180,E1 -3362.318,E2 -3362.318} C_VEL
LIN {X 0,Y 552.106,Z 470.837,A -85,B 0,C 180,E1 -3364.947,E2 -3364.947} C_VEL
LIN {X 0,Y 552.095,Z 470.829,A -85,B 0,C 180,E1 -3367.885,E2 -3367.885} C_VEL
LIN {X 0,Y 552.119,Z 470.831,A -85,B 0,C 180,E1 -3370.479,E2 -3370.479} C_VEL
LIN {X 0,Y 552.111,Z 470.835,A -85,B 0,C 180,E1 -3373.483,E2 -3373.483} C_VEL
LIN {X 0,Y 552.101,Z 470.834,A -85,B 0,C 180,E1 -3376.575,E2 -3376.575} C_VEL
LIN {X 0,Y 552.136,Z 470.834,A -85,B 0,C 180,E1 -3379.521,E2 -3379.521} C_VEL
LIN {X 0,Y 552.088,Z 470.832,A -85,B 0,C 180,E1 -3382.335,E2 -3382.335} C_VEL
LIN {X 0,Y 552.124,Z 470.835,A -85,B 0,C 180,E1 -3385.054,E2 -3385.054} C_VEL
LIN {X 0,Y 552.121,Z 470.833,A -85,B 0,C 180,E1 -3387.681,E2 -3387.681} C_VEL
LIN {X 0,Y 552.106,Z 470.832,A -85,B 0,C 180,E1 -3390.234,E2 -3390.234} C_VEL
LIN {X 0,Y 552.14,Z 470.828,A -85,B 0,C 180,E1 -3392.997,E2 -3392.997} C_VEL
LIN {X 0,Y 552.106,Z 470.837,A -85,B 0,C 180,E1 -3395.161,E2 -3395.161} C_VEL
LIN {X 0,Y 552.088,Z 470.838,A -85,B 0,C 180,E1 -3397.549,E2 -3397.549} C_VEL
LIN {X 0,Y 552.141,Z 470.825,A -85,B 0,C 180,E1 -3400.373,E2 -3400.373} C_VEL
LIN {X 0,Y 552.149,Z 470.829,A -85,B 0,C 180,E1 -3402.977,E2 -3402.977} C_VEL
LIN {X 0,Y 552.127,Z 470.825,A -85,B 0,C 180,E1 -3406.004,E2 -3406.004} C_VEL
LIN {X 0,Y 552.154,Z 470.827,A -85,B 0,C 180,E1 -3408.993,E2 -3408.993} C_VEL
LIN {X 0,Y 552.154,Z 470.826,A -85,B 0,C 180,E1 -3411.951,E2 -3411.951} C_VEL
LIN {X 0,Y 552.225,Z 470.812,A -85,B 0,C 180,E1 -3414.889,E2 -3414.889} C_VEL
LIN {X 0,Y 552.215,Z 470.822,A -85,B 0,C 180,E1 -3417.812,E2 -3417.812} C_VEL
LIN {X 0,Y 552.237,Z 470.813,A -85,B 0,C 180,E1 -3420.729,E2 -3420.729} C_VEL
LIN {X 0,Y 552.202,Z 470.816,A -85,B 0,C 180,E1 -3422.918,E2 -3422.918} C_VEL
LIN {X 0,Y 552.19,Z 470.826,A -85,B 0,C 180,E1 -3425.844,E2 -3425.844} C_VEL
LIN {X 0,Y 552.161,Z 470.822,A -85,B 0,C 180,E1 -3428.785,E2 -3428.785} C_VEL
LIN {X 0,Y 552.154,Z 470.832,A -85,B 0,C 180,E1 -3431.75,E2 -3431.75} C_VEL
LIN {X 0,Y 552.126,Z 470.829,A -85,B 0,C 180,E1 -3434.748,E2 -3434.748} C_VEL
LIN {X 0,Y 552.105,Z 470.836,A -85,B 0,C 180,E1 -3437.788,E2 -3437.788} C_VEL
LIN {X 0,Y 552.124,Z 470.832,A -85,B 0,C 180,E1 -3440.101,E2 -3440.101} C_VEL
LIN {X 0,Y 552.086,Z 470.833,A -85,B 0,C 180,E1 -3442.451,E2 -3442.451} C_VEL
LIN {X 0,Y 552.147,Z 470.828,A -85,B 0,C 180,E1 -3445.351,E2 -3445.351} C_VEL
LIN {X 0,Y 552.117,Z 470.833,A -85,B 0,C 180,E1 -3448.097,E2 -3448.097} C_VEL
LIN {X 0,Y 552.103,Z 470.828,A -85,B 0,C 180,E1 -3450.626,E2 -3450.626} C_VEL
LIN {X 0,Y 552.12,Z 470.832,A -85,B 0,C 180,E1 -3453.185,E2 -3453.185} C_VEL
LIN {X 0,Y 552.115,Z 470.832,A -85,B 0,C 180,E1 -3453.806,E2 -3453.806} C_VEL
LIN {X 0,Y 551.48,Z 470.914,A -85,B 0,C 180,E1 -3454.415,E2 -3454.415} C_VEL
LIN {X 0,Y 548.654,Z 471.266,A -85,B 0,C 180,E1 -3455.403,E2 -3455.403} C_VEL
LIN {X 0,Y 546.228,Z 471.565,A -85,B 0,C 180,E1 -3456.198,E2 -3456.198} C_VEL
LIN {X 0,Y 545.157,Z 471.696,A -85,B 0,C 180,E1 -3456.812,E2 -3456.812} C_VEL
LIN {X 0,Y 545.055,Z 471.709,A -85,B 0,C 180,E1 -3457.02,E2 -3457.02} C_VEL
LIN {X 0,Y 545.066,Z 471.709,A -85,B 0,C 180,E1 -3460.142,E2 -3460.142} C_VEL
LIN {X 0,Y 545.078,Z 471.709,A -85,B 0,C 180,E1 -3463.106,E2 -3463.106} C_VEL
LIN {X 0,Y 545.059,Z 471.701,A -85,B 0,C 180,E1 -3466.225,E2 -3466.225} C_VEL
LIN {X 0,Y 545.116,Z 471.701,A -85,B 0,C 180,E1 -3468.89,E2 -3468.89} C_VEL
LIN {X 0,Y 545.048,Z 471.717,A -85,B 0,C 180,E1 -3471.763,E2 -3471.763} C_VEL
LIN {X 0,Y 545.057,Z 471.71,A -85,B 0,C 180,E1 -3474.534,E2 -3474.534} C_VEL
LIN {X 0,Y 545.075,Z 471.71,A -85,B 0,C 180,E1 -3477.213,E2 -3477.213} C_VEL
LIN {X 0,Y 545.096,Z 471.715,A -85,B 0,C 180,E1 -3479.813,E2 -3479.813} C_VEL
LIN {X 0,Y 545.091,Z 471.707,A -85,B 0,C 180,E1 -3482.826,E2 -3482.826} C_VEL
LIN {X 0,Y 545.047,Z 471.718,A -85,B 0,C 180,E1 -3485.631,E2 -3485.631} C_VEL
LIN {X 0,Y 545.061,Z 471.71,A -85,B 0,C 180,E1 -3488.837,E2 -3488.837} C_VEL
LIN {X 0,Y 545.079,Z 471.709,A -85,B 0,C 180,E1 -3491.196,E2 -3491.196} C_VEL
LIN {X 0,Y 545.07,Z 471.714,A -85,B 0,C 180,E1 -3493.521,E2 -3493.521} C_VEL
LIN {X 0,Y 545.092,Z 471.715,A -85,B 0,C 180,E1 -3495.82,E2 -3495.82} C_VEL
LIN {X 0,Y 545.114,Z 471.704,A -85,B 0,C 180,E1 -3498.85,E2 -3498.85} C_VEL
LIN {X 0,Y 545.126,Z 471.711,A -85,B 0,C 180,E1 -3501.847,E2 -3501.847} C_VEL
LIN {X 0,Y 545.199,Z 471.694,A -85,B 0,C 180,E1 -3504.823,E2 -3504.823} C_VEL
LIN {X 0,Y 545.195,Z 471.701,A -85,B 0,C 180,E1 -3507.784,E2 -3507.784} C_VEL
LIN {X 0,Y 545.209,Z 471.694,A -85,B 0,C 180,E1 -3510.739,E2 -3510.739} C_VEL
LIN {X 0,Y 545.169,Z 471.698,A -85,B 0,C 180,E1 -3512.956,E2 -3512.956} C_VEL
LIN {X 0,Y 545.167,Z 471.705,A -85,B 0,C 180,E1 -3515.919,E2 -3515.919} C_VEL
LIN {X 0,Y 545.114,Z 471.704,A -85,B 0,C 180,E1 -3518.9,E2 -3518.9} C_VEL
LIN {X 0,Y 545.131,Z 471.709,A -85,B 0,C 180,E1 -3521.904,E2 -3521.904} C_VEL
LIN {X 0,Y 545.082,Z 471.709,A -85,B 0,C 180,E1 -3524.943,E2 -3524.943} C_VEL
LIN {X 0,Y 545.078,Z 471.717,A -85,B 0,C 180,E1 -3528.025,E2 -3528.025} C_VEL
LIN {X 0,Y 545.091,Z 471.712,A -85,B 0,C 180,E1 -3530.372,E2 -3530.372} C_VEL
LIN {X 0,Y 545.087,Z 471.709,A -85,B 0,C 180,E1 -3533.558,E2 -3533.558} C_VEL
LIN {X 0,Y 545.074,Z 471.717,A -85,B 0,C 180,E1 -3536,E2 -3536} C_VEL
LIN {X 0,Y 545.086,Z 471.709,A -85,B 0,C 180,E1 -3538.749,E2 -3538.749} C_VEL
LIN {X 0,Y 545.072,Z 471.711,A -85,B 0,C 180,E1 -3541.682,E2 -3541.682} C_VEL
LIN {X 0,Y 545.074,Z 471.711,A -85,B 0,C 180,E1 -3544.563,E2 -3544.563} C_VEL
LIN {X 0,Y 545.033,Z 471.708,A -85,B 0,C 180,E1 -3547.303,E2 -3547.303} C_VEL
LIN {X 0,Y 545.086,Z 471.716,A -85,B 0,C 180,E1 -3550.14,E2 -3550.14} C_VEL
LIN {X 0,Y 545.081,Z 471.696,A -85,B 0,C 180,E1 -3553.105,E2 -3553.105} C_VEL
LIN {X 0,Y 545.056,Z 471.718,A -85,B 0,C 180,E1 -3556.224,E2 -3556.224} C_VEL
LIN {X 0,Y 545.088,Z 471.705,A -85,B 0,C 180,E1 -3558.887,E2 -3558.887} C_VEL
LIN {X 0,Y 545.045,Z 471.714,A -85,B 0,C 180,E1 -3561.763,E2 -3561.763} C_VEL
LIN {X 0,Y 545.057,Z 471.715,A -85,B 0,C 180,E1 -3564.534,E2 -3564.534} C_VEL
LIN {X 0,Y 545.073,Z 471.708,A -85,B 0,C 180,E1 -3567.212,E2 -3567.212} C_VEL
LIN {X 0,Y 545.092,Z 471.704,A -85,B 0,C 180,E1 -3569.813,E2 -3569.813} C_VEL
LIN {X 0,Y 545.092,Z 471.708,A -85,B 0,C 180,E1 -3572.825,E2 -3572.825} C_VEL
LIN {X 0,Y 545.042,Z 471.708,A -85,B 0,C 180,E1 -3575.631,E2 -3575.631} C_VEL
LIN {X 0,Y 545.059,Z 471.713,A -85,B 0,C 180,E1 -3578.837,E2 -3578.837} C_VEL
LIN {X 0,Y 545.075,Z 471.705,A -85,B 0,C 180,E1 -3581.196,E2 -3581.196} C_VEL
LIN {X 0,Y 545.067,Z 471.705,A -85,B 0,C 180,E1 -3583.521,E2 -3583.521} C_VEL
LIN {X 0,Y 545.085,Z 471.708,A -85,B 0,C 180,E1 -3585.82,E2 -3585.82} C_VEL
LIN {X 0,Y 545.122,Z 471.7,A -85,B 0,C 180,E1 -3588.85,E2 -3588.85} C_VEL
LIN {X 0,Y 545.125,Z 471.7,A -85,B 0,C 180,E1 -3591.847,E2 -3591.847} C_VEL
LIN {X 0,Y 545.2,Z 471.695,A -85,B 0,C 180,E1 -3594.823,E2 -3594.823} C_VEL
LIN {X 0,Y 545.186,Z 471.688,A -85,B 0,C 180,E1 -3597.784,E2 -3597.784} C_VEL
LIN {X 0,Y 545.207,Z 471.697,A -85,B 0,C 180,E1 -3600.739,E2 -3600.739} C_VEL
LIN {X 0,Y 545.168,Z 471.697,A -85,B 0,C 180,E1 -3602.956,E2 -3602.956} C_VEL
LIN {X 0,Y 545.163,Z 471.691,A -85,B 0,C 180,E1 -3605.92,E2 -3605.92} C_VEL
LIN {X 0,Y 545.119,Z 471.706,A -85,B 0,C 180,E1 -3608.9,E2 -3608.9} C_VEL
LIN {X 0,Y 545.126,Z 471.701,A -85,B 0,C 180,E1 -3611.905,E2 -3611.905} C_VEL
LIN {X 0,Y 545.077,Z 471.71,A -85,B 0,C 180,E1 -3614.944,E2 -3614.944} C_VEL
LIN {X 0,Y 545.075,Z 471.709,A -85,B 0,C 180,E1 -3618.026,E2 -3618.026} C_VEL
LIN {X 0,Y 545.091,Z 471.709,A -85,B 0,C 180,E1 -3620.373,E2 -3620.373} C_VEL
LIN {X 0,Y 545.083,Z 471.706,A -85,B 0,C 180,E1 -3623.559,E2 -3623.559} C_VEL
LIN {X 0,Y 545.082,Z 471.707,A -85,B 0,C 180,E1 -3626.001,E2 -3626.001} C_VEL
LIN {X 0,Y 545.084,Z 471.715,A -85,B 0,C 180,E1 -3628.749,E2 -3628.749} C_VEL
LIN {X 0,Y 545.071,Z 471.707,A -85,B 0,C 180,E1 -3631.683,E2 -3631.683} C_VEL
LIN {X 0,Y 545.076,Z 471.713,A -85,B 0,C 180,E1 -3634.564,E2 -3634.564} C_VEL
LIN {X 0,Y 545.033,Z 471.712,A -85,B 0,C 180,E1 -3637.304,E2 -3637.304} C_VEL
LIN {X 0,Y 545.069,Z 471.711,A -85,B 0,C 180,E1 -3640.143,E2 -3640.143} C_VEL
LIN {X 0,Y 545.073,Z 471.713,A -85,B 0,C 180,E1 -3643.107,E2 -3643.107} C_VEL
LIN {X 0,Y 545.061,Z 471.709,A -85,B 0,C 180,E1 -3646.225,E2 -3646.225} C_VEL
LIN {X 0,Y 545.094,Z 471.714,A -85,B 0,C 180,E1 -3648.888,E2 -3648.888} C_VEL
LIN {X 0,Y 545.051,Z 471.704,A -85,B 0,C 180,E1 -3651.764,E2 -3651.764} C_VEL
LIN {X 0,Y 545.034,Z 471.705,A -85,B 0,C 180,E1 -3654.532,E2 -3654.532} C_VEL
LIN {X 0,Y 545.068,Z 471.711,A -85,B 0,C 180,E1 -3657.212,E2 -3657.212} C_VEL
LIN {X 0,Y 545.065,Z 471.708,A -85,B 0,C 180,E1 -3659.811,E2 -3659.811} C_VEL
LIN {X 0,Y 545.089,Z 471.701,A -85,B 0,C 180,E1 -3662.345,E2 -3662.345} C_VEL
LIN {X 0,Y 545.131,Z 471.895,A -85,B 0,C 180,E1 -3663.134,E2 -3663.134} C_VEL
LIN {X 0,Y 546.471,Z 479.547,A -85,B 0,C 180,E1 -3664.566,E2 -3664.566} C_VEL
LIN {X 0,Y 546.123,Z 497.768,A -85,B 0,C 180,E1 -3667.665,E2 -3667.665} C_VEL
LIN {X 0,Y 545.747,Z 514.388,A -85,B 0,C 180,E1 -3670.439,E2 -3670.439} C_VEL
LIN {X 0,Y 545.619,Z 526,A -85,B 0,C 180,E1 -3672.338,E2 -3672.338} C_VEL
LIN {X 0,Y 546.269,Z 529.512,A -85,B 0,C 180,E1 -3672.438,E2 -3672.438} C_VEL
LIN {X 0,Y 547.402,Z 535.271,A -85,B 0,C 180,E1 -3672.553,E2 -3672.553} C_VEL
LIN {X 0,Y 546.948,Z 661.185,A -85,B 0,C 180,E1 -3674.25,E2 -3674.25} C_VEL
LIN {X 0,Y 546.829,Z 672.117,A -85,B 0,C 180,E1 -3674.486,E2 -3674.486} C_VEL
LIN {X 0,Y 546.656,Z 682.726,A -85,B 0,C 180,E1 -3674.803,E2 -3674.803} C_VEL
LIN {X 0,Y 546.444,Z 693.914,A -85,B 0,C 180,E1 -3675.238,E2 -3675.238} C_VEL
LIN {X 0,Y 546.224,Z 704.529,A -85,B 0,C 180,E1 -3675.755,E2 -3675.755} C_VEL
LIN {X 0,Y 545.984,Z 714.144,A -85,B 0,C 180,E1 -3676.319,E2 -3676.319} C_VEL
LIN {X 0,Y 545.788,Z 723.615,A -85,B 0,C 180,E1 -3676.977,E2 -3676.977} C_VEL
LIN {X 0,Y 545.54,Z 732.813,A -85,B 0,C 180,E1 -3677.728,E2 -3677.728} C_VEL
LIN {X 0,Y 545.393,Z 740.847,A -85,B 0,C 180,E1 -3678.489,E2 -3678.489} C_VEL
LIN {X 0,Y 545.204,Z 749.249,A -85,B 0,C 180,E1 -3679.415,E2 -3679.415} C_VEL
LIN {X 0,Y 545.021,Z 756.508,A -85,B 0,C 180,E1 -3680.35,E2 -3680.35} C_VEL
LIN {X 0,Y 544.91,Z 762.742,A -85,B 0,C 180,E1 -3681.284,E2 -3681.284} C_VEL
LIN {X 0,Y 544.824,Z 768.114,A -85,B 0,C 180,E1 -3682.216,E2 -3682.216} C_VEL
LIN {X 0,Y 544.753,Z 773.846,A -85,B 0,C 180,E1 -3683.413,E2 -3683.413} C_VEL
LIN {X 0,Y 544.723,Z 777.909,A -85,B 0,C 180,E1 -3684.447,E2 -3684.447} C_VEL
LIN {X 0,Y 544.654,Z 781.427,A -85,B 0,C 180,E1 -3685.56,E2 -3685.56} C_VEL
LIN {X 0,Y 544.657,Z 783.325,A -85,B 0,C 180,E1 -3686.301,E2 -3686.301} C_VEL
LIN {X 0,Y 544.568,Z 785.996,A -85,B 0,C 180,E1 -3687.781,E2 -3687.781} C_VEL
LIN {X 0,Y 544.539,Z 787.277,A -85,B 0,C 180,E1 -3689.261,E2 -3689.261} C_VEL
LIN {X 0,Y 544.539,Z 787.5,A -85,B 0,C 180,E1 -3690,E2 -3690} C_VEL
LIN {X 0,Y 544.541,Z 786.802,A -85,B 0,C 180,E1 -3691.479,E2 -3691.479} C_VEL
LIN {X 0,Y 544.568,Z 785.996,A -85,B 0,C 180,E1 -3692.219,E2 -3692.219} C_VEL
LIN {X 0,Y 544.657,Z 783.325,A -85,B 0,C 180,E1 -3693.699,E2 -3693.699} C_VEL
LIN {X 0,Y 544.645,Z 779.165,A -85,B 0,C 180,E1 -3695.182,E2 -3695.182} C_VEL
LIN {X 0,Y 544.691,Z 775.017,A -85,B 0,C 180,E1 -3696.309,E2 -3696.309} C_VEL
LIN {X 0,Y 544.784,Z 770.014,A -85,B 0,C 180,E1 -3697.412,E2 -3697.412} C_VEL
LIN {X 0,Y 544.895,Z 763.872,A -85,B 0,C 180,E1 -3698.53,E2 -3698.53} C_VEL
LIN {X 0,Y 545.032,Z 757.838,A -85,B 0,C 180,E1 -3699.463,E2 -3699.463} C_VEL
LIN {X 0,Y 545.173,Z 750.804,A -85,B 0,C 180,E1 -3700.397,E2 -3700.397} C_VEL
LIN {X 0,Y 545.393,Z 742.651,A -85,B 0,C 180,E1 -3701.323,E2 -3701.323} C_VEL
LIN {X 0,Y 545.52,Z 733.869,A -85,B 0,C 180,E1 -3702.178,E2 -3702.178} C_VEL
LIN {X 0,Y 545.738,Z 724.852,A -85,B 0,C 180,E1 -3702.929,E2 -3702.929} C_VEL
LIN {X 0,Y 545.935,Z 715.605,A -85,B 0,C 180,E1 -3703.588,E2 -3703.588} C_VEL
LIN {X 0,Y 546.213,Z 706.28,A -85,B 0,C 180,E1 -3704.15,E2 -3704.15} C_VEL
LIN {X 0,Y 546.45,Z 694.986,A -85,B 0,C 180,E1 -3704.714,E2 -3704.714} C_VEL
LIN {X 0,Y 546.636,Z 684.665,A -85,B 0,C 180,E1 -3705.13,E2 -3705.13} C_VEL
LIN {X 0,Y 546.769,Z 673.345,A -85,B 0,C 180,E1 -3705.483,E2 -3705.483} C_VEL
LIN {X 0,Y 546.916,Z 662.543,A -85,B 0,C 180,E1 -3705.727,E2 -3705.727} C_VEL
LIN {X 0,Y 547.116,Z 628.811,A -85,B 0,C 180,E1 -3706.199,E2 -3706.199} C_VEL
LIN {X 0,Y 547.402,Z 535.221,A -85,B 0,C 180,E1 -3707.447,E2 -3707.447} C_VEL
LIN {X 0,Y 545.64,Z 526.302,A -85,B 0,C 180,E1 -3707.642,E2 -3707.642} C_VEL
LIN {X 0,Y 545.604,Z 523.731,A -85,B 0,C 180,E1 -3708.007,E2 -3708.007} C_VEL
LIN {X 0,Y 545.979,Z 504.979,A -85,B 0,C 180,E1 -3711.126,E2 -3711.126} C_VEL
LIN {X 0,Y 546.291,Z 487.827,A -85,B 0,C 180,E1 -3714.019,E2 -3714.019} C_VEL
LIN {X 0,Y 546.441,Z 479.585,A -85,B 0,C 180,E1 -3715.433,E2 -3715.433} C_VEL
LIN {X 0,Y 545.131,Z 471.868,A -85,B 0,C 180,E1 -3716.866,E2 -3716.866} C_VEL
LIN {X 0,Y 545.064,Z 471.716,A -85,B 0,C 180,E1 -3719.338,E2 -3719.338} C_VEL
LIN {X 0,Y 545.066,Z 471.708,A -85,B 0,C 180,E1 -3721.913,E2 -3721.913} C_VEL
LIN {X 0,Y 545.07,Z 471.711,A -85,B 0,C 180,E1 -3724.563,E2 -3724.563} C_VEL
LIN {X 0,Y 545.034,Z 471.705,A -85,B 0,C 180,E1 -3727.303,E2 -3727.303} C_VEL
LIN {X 0,Y 545.072,Z 471.709,A -85,B 0,C 180,E1 -3730.141,E2 -3730.141} C_VEL
LIN {X 0,Y 545.083,Z 471.709,A -85,B 0,C 180,E1 -3733.105,E2 -3733.105} C_VEL
LIN {X 0,Y 545.046,Z 471.712,A -85,B 0,C 180,E1 -3736.225,E2 -3736.225} C_VEL
LIN {X 0,Y 545.091,Z 471.708,A -85,B 0,C 180,E1 -3738.886,E2 -3738.886} C_VEL
LIN {X 0,Y 545.048,Z 471.712,A -85,B 0,C 180,E1 -3741.762,E2 -3741.762} C_VEL
LIN {X 0,Y 545.06,Z 471.71,A -85,B 0,C 180,E1 -3744.533,E2 -3744.533} C_VEL
LIN {X 0,Y 545.075,Z 471.712,A -85,B 0,C 180,E1 -3747.212,E2 -3747.212} C_VEL
LIN {X 0,Y 545.059,Z 471.712,A -85,B 0,C 180,E1 -3749.81,E2 -3749.81} C_VEL
LIN {X 0,Y 545.089,Z 471.702,A -85,B 0,C 180,E1 -3752.344,E2 -3752.344} C_VEL
LIN {X 0,Y 545.111,Z 471.704,A -85,B 0,C 180,E1 -3754.82,E2 -3754.82} C_VEL
LIN {X 0,Y 545.037,Z 471.72,A -85,B 0,C 180,E1 -3757.242,E2 -3757.242} C_VEL
LIN {X 0,Y 545.113,Z 471.7,A -85,B 0,C 180,E1 -3760.414,E2 -3760.414} C_VEL
LIN {X 0,Y 545.068,Z 471.715,A -85,B 0,C 180,E1 -3763.521,E2 -3763.521} C_VEL
LIN {X 0,Y 545.086,Z 471.704,A -85,B 0,C 180,E1 -3765.819,E2 -3765.819} C_VEL
LIN {X 0,Y 545.109,Z 471.703,A -85,B 0,C 180,E1 -3768.849,E2 -3768.849} C_VEL
LIN {X 0,Y 545.125,Z 471.703,A -85,B 0,C 180,E1 -3771.847,E2 -3771.847} C_VEL
LIN {X 0,Y 545.199,Z 471.686,A -85,B 0,C 180,E1 -3774.823,E2 -3774.823} C_VEL
LIN {X 0,Y 545.187,Z 471.698,A -85,B 0,C 180,E1 -3777.783,E2 -3777.783} C_VEL
LIN {X 0,Y 545.207,Z 471.688,A -85,B 0,C 180,E1 -3780.738,E2 -3780.738} C_VEL
LIN {X 0,Y 545.168,Z 471.692,A -85,B 0,C 180,E1 -3782.955,E2 -3782.955} C_VEL
LIN {X 0,Y 545.162,Z 471.7,A -85,B 0,C 180,E1 -3785.919,E2 -3785.919} C_VEL
LIN {X 0,Y 545.118,Z 471.7,A -85,B 0,C 180,E1 -3788.9,E2 -3788.9} C_VEL
LIN {X 0,Y 545.126,Z 471.705,A -85,B 0,C 180,E1 -3791.904,E2 -3791.904} C_VEL
LIN {X 0,Y 545.075,Z 471.709,A -85,B 0,C 180,E1 -3794.943,E2 -3794.943} C_VEL
LIN {X 0,Y 545.073,Z 471.708,A -85,B 0,C 180,E1 -3798.026,E2 -3798.026} C_VEL
LIN {X 0,Y 545.089,Z 471.706,A -85,B 0,C 180,E1 -3800.372,E2 -3800.372} C_VEL
LIN {X 0,Y 545.081,Z 471.712,A -85,B 0,C 180,E1 -3803.559,E2 -3803.559} C_VEL
LIN {X 0,Y 545.079,Z 471.711,A -85,B 0,C 180,E1 -3806,E2 -3806} C_VEL
LIN {X 0,Y 545.083,Z 471.706,A -85,B 0,C 180,E1 -3808.749,E2 -3808.749} C_VEL
LIN {X 0,Y 545.069,Z 471.715,A -85,B 0,C 180,E1 -3811.683,E2 -3811.683} C_VEL
LIN {X 0,Y 545.076,Z 471.707,A -85,B 0,C 180,E1 -3814.563,E2 -3814.563} C_VEL
LIN {X 0,Y 545.055,Z 471.709,A -85,B 0,C 180,E1 -3817.02,E2 -3817.02} C_VEL
LIN {X 0,Y 544.348,Z 471.805,A -85,B 0,C 180,E1 -3817.637,E2 -3817.637} C_VEL
LIN {X 0,Y 541.485,Z 472.161,A -85,B 0,C 180,E1 -3818.638,E2 -3818.638} C_VEL
LIN {X 0,Y 539.099,Z 472.458,A -85,B 0,C 180,E1 -3819.444,E2 -3819.444} C_VEL
LIN {X 0,Y 538.089,Z 472.58,A -85,B 0,C 180,E1 -3820.066,E2 -3820.066} C_VEL
LIN {X 0,Y 538.014,Z 472.586,A -85,B 0,C 180,E1 -3820.276,E2 -3820.276} C_VEL
LIN {X 0,Y 538.024,Z 472.587,A -85,B 0,C 180,E1 -3822.989,E2 -3822.989} C_VEL
LIN {X 0,Y 538.022,Z 472.582,A -85,B 0,C 180,E1 -3825.926,E2 -3825.926} C_VEL
LIN {X 0,Y 538.073,Z 472.58,A -85,B 0,C 180,E1 -3829.249,E2 -3829.249} C_VEL
LIN {X 0,Y 537.988,Z 472.589,A -85,B 0,C 180,E1 -3832.123,E2 -3832.123} C_VEL
LIN {X 0,Y 538.013,Z 472.587,A -85,B 0,C 180,E1 -3834.918,E2 -3834.918} C_VEL
LIN {X 0,Y 538.025,Z 472.593,A -85,B 0,C 180,E1 -3837.619,E2 -3837.619} C_VEL
LIN {X 0,Y 538.037,Z 472.589,A -85,B 0,C 180,E1 -3840.241,E2 -3840.241} C_VEL
LIN {X 0,Y 538.061,Z 472.583,A -85,B 0,C 180,E1 -3842.797,E2 -3842.797} C_VEL
LIN {X 0,Y 538.044,Z 472.587,A -85,B 0,C 180,E1 -3845.293,E2 -3845.293} C_VEL
LIN {X 0,Y 538.011,Z 472.596,A -85,B 0,C 180,E1 -3848.042,E2 -3848.042} C_VEL
LIN {X 0,Y 538.035,Z 472.586,A -85,B 0,C 180,E1 -3850.94,E2 -3850.94} C_VEL
LIN {X 0,Y 538.021,Z 472.59,A -85,B 0,C 180,E1 -3853.299,E2 -3853.299} C_VEL
LIN {X 0,Y 538.06,Z 472.588,A -85,B 0,C 180,E1 -3855.631,E2 -3855.631} C_VEL
LIN {X 0,Y 538.073,Z 472.582,A -85,B 0,C 180,E1 -3858.702,E2 -3858.702} C_VEL
LIN {X 0,Y 538.083,Z 472.586,A -85,B 0,C 180,E1 -3861.74,E2 -3861.74} C_VEL
LIN {X 0,Y 538.157,Z 472.572,A -85,B 0,C 180,E1 -3864.755,E2 -3864.755} C_VEL
LIN {X 0,Y 538.166,Z 472.576,A -85,B 0,C 180,E1 -3867.755,E2 -3867.755} C_VEL
LIN {X 0,Y 538.179,Z 472.57,A -85,B 0,C 180,E1 -3870.748,E2 -3870.748} C_VEL
LIN {X 0,Y 538.135,Z 472.574,A -85,B 0,C 180,E1 -3872.994,E2 -3872.994} C_VEL
LIN {X 0,Y 538.12,Z 472.583,A -85,B 0,C 180,E1 -3875.997,E2 -3875.997} C_VEL
LIN {X 0,Y 538.065,Z 472.582,A -85,B 0,C 180,E1 -3879.017,E2 -3879.017} C_VEL
LIN {X 0,Y 538.08,Z 472.588,A -85,B 0,C 180,E1 -3882.062,E2 -3882.062} C_VEL
LIN {X 0,Y 538.042,Z 472.586,A -85,B 0,C 180,E1 -3885.144,E2 -3885.144} C_VEL
LIN {X 0,Y 538.03,Z 472.594,A -85,B 0,C 180,E1 -3888.27,E2 -3888.27} C_VEL
LIN {X 0,Y 538.035,Z 472.588,A -85,B 0,C 180,E1 -3890.651,E2 -3890.651} C_VEL
LIN {X 0,Y 538.019,Z 472.594,A -85,B 0,C 180,E1 -3893.887,E2 -3893.887} C_VEL
LIN {X 0,Y 538.037,Z 472.592,A -85,B 0,C 180,E1 -3896.366,E2 -3896.366} C_VEL
LIN {X 0,Y 538.051,Z 472.584,A -85,B 0,C 180,E1 -3898.938,E2 -3898.938} C_VEL
LIN {X 0,Y 538.022,Z 472.592,A -85,B 0,C 180,E1 -3901.89,E2 -3901.89} C_VEL
LIN {X 0,Y 538.024,Z 472.589,A -85,B 0,C 180,E1 -3904.62,E2 -3904.62} C_VEL
LIN {X 0,Y 538.001,Z 472.583,A -85,B 0,C 180,E1 -3907.17,E2 -3907.17} C_VEL
LIN {X 0,Y 538.047,Z 472.587,A -85,B 0,C 180,E1 -3909.794,E2 -3909.794} C_VEL
LIN {X 0,Y 538.017,Z 472.576,A -85,B 0,C 180,E1 -3912.785,E2 -3912.785} C_VEL
LIN {X 0,Y 538.02,Z 472.589,A -85,B 0,C 180,E1 -3915.925,E2 -3915.925} C_VEL
LIN {X 0,Y 538.043,Z 472.581,A -85,B 0,C 180,E1 -3919.224,E2 -3919.224} C_VEL
LIN {X 0,Y 537.985,Z 472.599,A -85,B 0,C 180,E1 -3922.122,E2 -3922.122} C_VEL
LIN {X 0,Y 538.013,Z 472.588,A -85,B 0,C 180,E1 -3924.917,E2 -3924.917} C_VEL
LIN {X 0,Y 538.023,Z 472.587,A -85,B 0,C 180,E1 -3927.618,E2 -3927.618} C_VEL
LIN {X 0,Y 538.034,Z 472.588,A -85,B 0,C 180,E1 -3930.24,E2 -3930.24} C_VEL
LIN {X 0,Y 538.061,Z 472.584,A -85,B 0,C 180,E1 -3932.797,E2 -3932.797} C_VEL
LIN {X 0,Y 538.039,Z 472.579,A -85,B 0,C 180,E1 -3935.293,E2 -3935.293} C_VEL
LIN {X 0,Y 538.005,Z 472.591,A -85,B 0,C 180,E1 -3938.042,E2 -3938.042} C_VEL
LIN {X 0,Y 538.03,Z 472.584,A -85,B 0,C 180,E1 -3940.94,E2 -3940.94} C_VEL
LIN {X 0,Y 538.017,Z 472.583,A -85,B 0,C 180,E1 -3943.299,E2 -3943.299} C_VEL
LIN {X 0,Y 538.053,Z 472.582,A -85,B 0,C 180,E1 -3945.631,E2 -3945.631} C_VEL
LIN {X 0,Y 538.079,Z 472.579,A -85,B 0,C 180,E1 -3948.702,E2 -3948.702} C_VEL
LIN {X 0,Y 538.081,Z 472.576,A -85,B 0,C 180,E1 -3951.74,E2 -3951.74} C_VEL
LIN {X 0,Y 538.175,Z 472.571,A -85,B 0,C 180,E1 -3954.756,E2 -3954.756} C_VEL
LIN {X 0,Y 538.158,Z 472.563,A -85,B 0,C 180,E1 -3957.755,E2 -3957.755} C_VEL
LIN {X 0,Y 538.177,Z 472.572,A -85,B 0,C 180,E1 -3960.749,E2 -3960.749} C_VEL
LIN {X 0,Y 538.134,Z 472.573,A -85,B 0,C 180,E1 -3962.995,E2 -3962.995} C_VEL
LIN {X 0,Y 538.115,Z 472.569,A -85,B 0,C 180,E1 -3965.998,E2 -3965.998} C_VEL
LIN {X 0,Y 538.068,Z 472.583,A -85,B 0,C 180,E1 -3969.018,E2 -3969.018} C_VEL
LIN {X 0,Y 538.074,Z 472.581,A -85,B 0,C 180,E1 -3972.063,E2 -3972.063} C_VEL
LIN {X 0,Y 538.037,Z 472.585,A -85,B 0,C 180,E1 -3975.144,E2 -3975.144} C_VEL
LIN {X 0,Y 538.027,Z 472.59,A -85,B 0,C 180,E1 -3978.271,E2 -3978.271} C_VEL
LIN {X 0,Y 538.034,Z 472.588,A -85,B 0,C 180,E1 -3980.652,E2 -3980.652} C_VEL
LIN {X 0,Y 538.016,Z 472.588,A -85,B 0,C 180,E1 -3983.888,E2 -3983.888} C_VEL
LIN {X 0,Y 538.043,Z 472.588,A -85,B 0,C 180,E1 -3986.367,E2 -3986.367} C_VEL
LIN {X 0,Y 538.025,Z 472.591,A -85,B 0,C 180,E1 -3988.935,E2 -3988.935} C_VEL
LIN {X 0,Y 538.021,Z 472.586,A -85,B 0,C 180,E1 -3991.891,E2 -3991.891} C_VEL
LIN {X 0,Y 538.026,Z 472.592,A -85,B 0,C 180,E1 -3994.622,E2 -3994.622} C_VEL
LIN {X 0,Y 538.002,Z 472.589,A -85,B 0,C 180,E1 -3997.171,E2 -3997.171} C_VEL
LIN {X 0,Y 538.024,Z 472.587,A -85,B 0,C 180,E1 -3999.797,E2 -3999.797} C_VEL
LIN {X 0,Y 538.028,Z 472.584,A -85,B 0,C 180,E1 -4001.88,E2 -4001.88} C_VEL
LIN {X 0,Y 538.028,Z 472.586,A -85,B 0,C 180,E1 -4005.141,E2 -4005.141} C_VEL
LIN {X 0,Y 538.038,Z 472.584,A -85,B 0,C 180,E1 -4008.229,E2 -4008.229} C_VEL
LIN {X 0,Y 538.013,Z 472.584,A -85,B 0,C 180,E1 -4011.171,E2 -4011.171} C_VEL
LIN {X 0,Y 537.991,Z 472.576,A -85,B 0,C 180,E1 -4014.089,E2 -4014.089} C_VEL
LIN {X 0,Y 538.028,Z 472.596,A -85,B 0,C 180,E1 -4016.728,E2 -4016.728} C_VEL
LIN {X 0,Y 538.026,Z 472.582,A -85,B 0,C 180,E1 -4019.557,E2 -4019.557} C_VEL
LIN {X 0,Y 538.044,Z 472.583,A -85,B 0,C 180,E1 -4021.951,E2 -4021.951} C_VEL
LIN {X 0,Y 538.072,Z 472.692,A -85,B 0,C 180,E1 -4022.902,E2 -4022.902} C_VEL
LIN {X 0,Y 539.435,Z 479.925,A -85,B 0,C 180,E1 -4024.306,E2 -4024.306} C_VEL
LIN {X 0,Y 539.309,Z 490.682,A -85,B 0,C 180,E1 -4026.174,E2 -4026.174} C_VEL
LIN {X 0,Y 538.976,Z 508.35,A -85,B 0,C 180,E1 -4029.187,E2 -4029.187} C_VEL
LIN {X 0,Y 538.626,Z 525.979,A -85,B 0,C 180,E1 -4032.106,E2 -4032.106} C_VEL
LIN {X 0,Y 540.233,Z 534.081,A -85,B 0,C 180,E1 -4032.299,E2 -4032.299} C_VEL
LIN {X 0,Y 540.691,Z 537.749,A -85,B 0,C 180,E1 -4032.364,E2 -4032.364} C_VEL
LIN {X 0,Y 540.12,Z 661.136,A -85,B 0,C 180,E1 -4034.046,E2 -4034.046} C_VEL
LIN {X 0,Y 539.97,Z 671.811,A -85,B 0,C 180,E1 -4034.277,E2 -4034.277} C_VEL
LIN {X 0,Y 539.826,Z 681.397,A -85,B 0,C 180,E1 -4034.559,E2 -4034.559} C_VEL
LIN {X 0,Y 539.576,Z 692.822,A -85,B 0,C 180,E1 -4034.997,E2 -4034.997} C_VEL
LIN {X 0,Y 539.378,Z 702.768,A -85,B 0,C 180,E1 -4035.474,E2 -4035.474} C_VEL
LIN {X 0,Y 539.1,Z 712.669,A -85,B 0,C 180,E1 -4036.044,E2 -4036.044} C_VEL
LIN {X 0,Y 538.88,Z 722.366,A -85,B 0,C 180,E1 -4036.711,E2 -4036.711} C_VEL
LIN {X 0,Y 538.619,Z 731.749,A -85,B 0,C 180,E1 -4037.472,E2 -4037.472} C_VEL
LIN {X 0,Y 538.418,Z 739.834,A -85,B 0,C 180,E1 -4038.232,E2 -4038.232} C_VEL
LIN {X 0,Y 538.229,Z 747.685,A -85,B 0,C 180,E1 -4039.086,E2 -4039.086} C_VEL
LIN {X 0,Y 538.022,Z 755.169,A -85,B 0,C 180,E1 -4040.033,E2 -4040.033} C_VEL
LIN {X 0,Y 537.861,Z 762.735,A -85,B 0,C 180,E1 -4041.169,E2 -4041.169} C_VEL
LIN {X 0,Y 537.765,Z 768.106,A -85,B 0,C 180,E1 -4042.113,E2 -4042.113} C_VEL
LIN {X 0,Y 537.666,Z 773.498,A -85,B 0,C 180,E1 -4043.244,E2 -4043.244} C_VEL
LIN {X 0,Y 537.653,Z 777.904,A -85,B 0,C 180,E1 -4044.374,E2 -4044.374} C_VEL
LIN {X 0,Y 537.549,Z 781.42,A -85,B 0,C 180,E1 -4045.501,E2 -4045.501} C_VEL
LIN {X 0,Y 537.576,Z 783.326,A -85,B 0,C 180,E1 -4046.252,E2 -4046.252} C_VEL
LIN {X 0,Y 537.487,Z 785.991,A -85,B 0,C 180,E1 -4047.752,E2 -4047.752} C_VEL
LIN {X 0,Y 537.439,Z 787.27,A -85,B 0,C 180,E1 -4049.251,E2 -4049.251} C_VEL
LIN {X 0,Y 537.44,Z 787.5,A -85,B 0,C 180,E1 -4050,E2 -4050} C_VEL
LIN {X 0,Y 537.446,Z 786.799,A -85,B 0,C 180,E1 -4051.499,E2 -4051.499} C_VEL
LIN {X 0,Y 537.487,Z 785.991,A -85,B 0,C 180,E1 -4052.248,E2 -4052.248} C_VEL
LIN {X 0,Y 537.576,Z 783.326,A -85,B 0,C 180,E1 -4053.748,E2 -4053.748} C_VEL
LIN {X 0,Y 537.578,Z 779.159,A -85,B 0,C 180,E1 -4055.251,E2 -4055.251} C_VEL
LIN {X 0,Y 537.601,Z 775.437,A -85,B 0,C 180,E1 -4056.29,E2 -4056.29} C_VEL
LIN {X 0,Y 537.704,Z 770.006,A -85,B 0,C 180,E1 -4057.51,E2 -4057.51} C_VEL
LIN {X 0,Y 537.825,Z 763.866,A -85,B 0,C 180,E1 -4058.643,E2 -4058.643} C_VEL
LIN {X 0,Y 537.966,Z 757.83,A -85,B 0,C 180,E1 -4059.588,E2 -4059.588} C_VEL
LIN {X 0,Y 538.164,Z 750.794,A -85,B 0,C 180,E1 -4060.534,E2 -4060.534} C_VEL
LIN {X 0,Y 538.37,Z 743,A -85,B 0,C 180,E1 -4061.435,E2 -4061.435} C_VEL
LIN {X 0,Y 538.537,Z 733.861,A -85,B 0,C 180,E1 -4062.339,E2 -4062.339} C_VEL
LIN {X 0,Y 538.796,Z 724.839,A -85,B 0,C 180,E1 -4063.099,E2 -4063.099} C_VEL
LIN {X 0,Y 539.012,Z 715.591,A -85,B 0,C 180,E1 -4063.766,E2 -4063.766} C_VEL
LIN {X 0,Y 539.307,Z 706.269,A -85,B 0,C 180,E1 -4064.335,E2 -4064.335} C_VEL
LIN {X 0,Y 539.573,Z 694.966,A -85,B 0,C 180,E1 -4064.906,E2 -4064.906} C_VEL
LIN {X 0,Y 539.769,Z 685.357,A -85,B 0,C 180,E1 -4065.302,E2 -4065.302} C_VEL
LIN {X 0,Y 539.92,Z 673.774,A -85,B 0,C 180,E1 -4065.673,E2 -4065.673} C_VEL
LIN {X 0,Y 540.088,Z 662.495,A -85,B 0,C 180,E1 -4065.931,E2 -4065.931} C_VEL
LIN {X 0,Y 540.297,Z 630.6,A -85,B 0,C 180,E1 -4066.385,E2 -4066.385} C_VEL
LIN {X 0,Y 540.614,Z 536.036,A -85,B 0,C 180,E1 -4067.662,E2 -4067.662} C_VEL
LIN {X 0,Y 538.653,Z 526.228,A -85,B 0,C 180,E1 -4067.877,E2 -4067.877} C_VEL
LIN {X 0,Y 538.622,Z 524.849,A -85,B 0,C 180,E1 -4068.045,E2 -4068.045} C_VEL
LIN {X 0,Y 539.035,Z 504.819,A -85,B 0,C 180,E1 -4071.411,E2 -4071.411} C_VEL
LIN {X 0,Y 539.372,Z 488.493,A -85,B 0,C 180,E1 -4074.203,E2 -4074.203} C_VEL
LIN {X 0,Y 539.418,Z 479.965,A -85,B 0,C 180,E1 -4075.697,E2 -4075.697} C_VEL
LIN {X 0,Y 538.072,Z 472.654,A -85,B 0,C 180,E1 -4077.098,E2 -4077.098} C_VEL
LIN {X 0,Y 538.018,Z 472.588,A -85,B 0,C 180,E1 -4079.76,E2 -4079.76} C_VEL
LIN {X 0,Y 538.023,Z 472.585,A -85,B 0,C 180,E1 -4082.382,E2 -4082.382} C_VEL
LIN {X 0,Y 537.999,Z 472.587,A -85,B 0,C 180,E1 -4085.083,E2 -4085.083} C_VEL
LIN {X 0,Y 537.991,Z 472.585,A -85,B 0,C 180,E1 -4087.877,E2 -4087.877} C_VEL
LIN {X 0,Y 538.049,Z 472.586,A -85,B 0,C 180,E1 -4090.775,E2 -4090.775} C_VEL
LIN {X 0,Y 538.025,Z 472.583,A -85,B 0,C 180,E1 -4094.074,E2 -4094.074} C_VEL
LIN {X 0,Y 538.014,Z 472.596,A -85,B 0,C 180,E1 -4097.213,E2 -4097.213} C_VEL
LIN {X 0,Y 538.073,Z 472.588,A -85,B 0,C 180,E1 -4099.248,E2 -4099.248} C_VEL
LIN {X 0,Y 537.988,Z 472.588,A -85,B 0,C 180,E1 -4102.122,E2 -4102.122} C_VEL
LIN {X 0,Y 538.015,Z 472.591,A -85,B 0,C 180,E1 -4104.917,E2 -4104.917} C_VEL
LIN {X 0,Y 538.025,Z 472.59,A -85,B 0,C 180,E1 -4107.617,E2 -4107.617} C_VEL
LIN {X 0,Y 538.012,Z 472.588,A -85,B 0,C 180,E1 -4110.238,E2 -4110.238} C_VEL
LIN {X 0,Y 538.064,Z 472.579,A -85,B 0,C 180,E1 -4112.796,E2 -4112.796} C_VEL
LIN {X 0,Y 538.042,Z 472.591,A -85,B 0,C 180,E1 -4115.292,E2 -4115.292} C_VEL
LIN {X 0,Y 538.007,Z 472.586,A -85,B 0,C 180,E1 -4118.041,E2 -4118.041} C_VEL
LIN {X 0,Y 538.033,Z 472.585,A -85,B 0,C 180,E1 -4120.94,E2 -4120.94} C_VEL
LIN {X 0,Y 538.019,Z 472.594,A -85,B 0,C 180,E1 -4123.299,E2 -4123.299} C_VEL
LIN {X 0,Y 538.055,Z 472.582,A -85,B 0,C 180,E1 -4125.63,E2 -4125.63} C_VEL
LIN {X 0,Y 538.068,Z 472.579,A -85,B 0,C 180,E1 -4128.701,E2 -4128.701} C_VEL
LIN {X 0,Y 538.081,Z 472.582,A -85,B 0,C 180,E1 -4131.739,E2 -4131.739} C_VEL
LIN {X 0,Y 538.156,Z 472.563,A -85,B 0,C 180,E1 -4134.755,E2 -4134.755} C_VEL
LIN {X 0,Y 538.158,Z 472.574,A -85,B 0,C 180,E1 -4137.754,E2 -4137.754} C_VEL
LIN {X 0,Y 538.176,Z 472.564,A -85,B 0,C 180,E1 -4140.748,E2 -4140.748} C_VEL
LIN {X 0,Y 538.134,Z 472.568,A -85,B 0,C 180,E1 -4142.994,E2 -4142.994} C_VEL
LIN {X 0,Y 538.114,Z 472.577,A -85,B 0,C 180,E1 -4145.997,E2 -4145.997} C_VEL
LIN {X 0,Y 538.067,Z 472.579,A -85,B 0,C 180,E1 -4149.017,E2 -4149.017} C_VEL
LIN {X 0,Y 538.074,Z 472.582,A -85,B 0,C 180,E1 -4152.062,E2 -4152.062} C_VEL
LIN {X 0,Y 538.035,Z 472.587,A -85,B 0,C 180,E1 -4155.144,E2 -4155.144} C_VEL
LIN {X 0,Y 538.025,Z 472.584,A -85,B 0,C 180,E1 -4158.27,E2 -4158.27} C_VEL
LIN {X 0,Y 538.032,Z 472.585,A -85,B 0,C 180,E1 -4160.651,E2 -4160.651} C_VEL
LIN {X 0,Y 538.014,Z 472.588,A -85,B 0,C 180,E1 -4163.887,E2 -4163.887} C_VEL
LIN {X 0,Y 538.04,Z 472.584,A -85,B 0,C 180,E1 -4166.366,E2 -4166.366} C_VEL
LIN {X 0,Y 538.046,Z 472.583,A -85,B 0,C 180,E1 -4168.939,E2 -4168.939} C_VEL
LIN {X 0,Y 538.019,Z 472.593,A -85,B 0,C 180,E1 -4171.891,E2 -4171.891} C_VEL
LIN {X 0,Y 538.026,Z 472.585,A -85,B 0,C 180,E1 -4174.622,E2 -4174.622} C_VEL
LIN {X 0,Y 537.999,Z 472.589,A -85,B 0,C 180,E1 -4177.171,E2 -4177.171} C_VEL
LIN {X 0,Y 538.014,Z 472.586,A -85,B 0,C 180,E1 -4180.276,E2 -4180.276} C_VEL
LIN {X 0,Y 537.364,Z 472.666,A -85,B 0,C 180,E1 -4180.901,E2 -4180.901} C_VEL
LIN {X 0,Y 534.513,Z 473.031,A -85,B 0,C 180,E1 -4181.916,E2 -4181.916} C_VEL
LIN {X 0,Y 532.09,Z 473.337,A -85,B 0,C 180,E1 -4182.733,E2 -4182.733} C_VEL
LIN {X 0,Y 531.042,Z 473.464,A -85,B 0,C 180,E1 -4183.364,E2 -4183.364} C_VEL
LIN {X 0,Y 530.954,Z 473.472,A -85,B 0,C 180,E1 -4183.578,E2 -4183.578} C_VEL
LIN {X 0,Y 530.96,Z 473.453,A -85,B 0,C 180,E1 -4186.506,E2 -4186.506} C_VEL
LIN {X 0,Y 531.02,Z 473.463,A -85,B 0,C 180,E1 -4189.572,E2 -4189.572} C_VEL
LIN {X 0,Y 530.962,Z 473.46,A -85,B 0,C 180,E1 -4192.577,E2 -4192.577} C_VEL
LIN {X 0,Y 530.994,Z 473.464,A -85,B 0,C 180,E1 -4195.311,E2 -4195.311} C_VEL
LIN {X 0,Y 530.977,Z 473.471,A -85,B 0,C 180,E1 -4198.033,E2 -4198.033} C_VEL
LIN {X 0,Y 531.002,Z 473.462,A -85,B 0,C 180,E1 -4200.871,E2 -4200.871} C_VEL
LIN {X 0,Y 531,Z 473.464,A -85,B 0,C 180,E1 -4203.257,E2 -4203.257} C_VEL
LIN {X 0,Y 530.992,Z 473.471,A -85,B 0,C 180,E1 -4205.958,E2 -4205.958} C_VEL
LIN {X 0,Y 530.995,Z 473.463,A -85,B 0,C 180,E1 -4209.062,E2 -4209.062} C_VEL
LIN {X 0,Y 531.012,Z 473.465,A -85,B 0,C 180,E1 -4212.278,E2 -4212.278} C_VEL
LIN {X 0,Y 531.015,Z 473.464,A -85,B 0,C 180,E1 -4215.436,E2 -4215.436} C_VEL
LIN {X 0,Y 531.033,Z 473.46,A -85,B 0,C 180,E1 -4218.55,E2 -4218.55} C_VEL
LIN {X 0,Y 531.052,Z 473.461,A -85,B 0,C 180,E1 -4221.63,E2 -4221.63} C_VEL
LIN {X 0,Y 531.116,Z 473.449,A -85,B 0,C 180,E1 -4224.685,E2 -4224.685} C_VEL
LIN {X 0,Y 531.138,Z 473.452,A -85,B 0,C 180,E1 -4227.725,E2 -4227.725} C_VEL
LIN {X 0,Y 531.149,Z 473.445,A -85,B 0,C 180,E1 -4230.758,E2 -4230.758} C_VEL
LIN {X 0,Y 531.102,Z 473.451,A -85,B 0,C 180,E1 -4233.034,E2 -4233.034} C_VEL
LIN {X 0,Y 531.08,Z 473.46,A -85,B 0,C 180,E1 -4236.077,E2 -4236.077} C_VEL
LIN {X 0,Y 531.025,Z 473.46,A -85,B 0,C 180,E1 -4239.138,E2 -4239.138} C_VEL
LIN {X 0,Y 531.037,Z 473.465,A -85,B 0,C 180,E1 -4242.225,E2 -4242.225} C_VEL
LIN {X 0,Y 530.992,Z 473.465,A -85,B 0,C 180,E1 -4245.349,E2 -4245.349} C_VEL
LIN {X 0,Y 530.989,Z 473.468,A -85,B 0,C 180,E1 -4248.521,E2 -4248.521} C_VEL
LIN {X 0,Y 530.995,Z 473.463,A -85,B 0,C 180,E1 -4250.938,E2 -4250.938} C_VEL
LIN {X 0,Y 530.975,Z 473.473,A -85,B 0,C 180,E1 -4254.224,E2 -4254.224} C_VEL
LIN {X 0,Y 531,Z 473.464,A -85,B 0,C 180,E1 -4256.743,E2 -4256.743} C_VEL
LIN {X 0,Y 530.995,Z 473.463,A -85,B 0,C 180,E1 -4259.321,E2 -4259.321} C_VEL
LIN {X 0,Y 530.974,Z 473.473,A -85,B 0,C 180,E1 -4262.103,E2 -4262.103} C_VEL
LIN {X 0,Y 530.981,Z 473.464,A -85,B 0,C 180,E1 -4264.854,E2 -4264.854} C_VEL
LIN {X 0,Y 530.96,Z 473.461,A -85,B 0,C 180,E1 -4267.507,E2 -4267.507} C_VEL
LIN {X 0,Y 531.019,Z 473.463,A -85,B 0,C 180,E1 -4270.428,E2 -4270.428} C_VEL
LIN {X 0,Y 530.96,Z 473.453,A -85,B 0,C 180,E1 -4273.494,E2 -4273.494} C_VEL
LIN {X 0,Y 530.957,Z 473.473,A -85,B 0,C 180,E1 -4276.505,E2 -4276.505} C_VEL
LIN {X 0,Y 530.98,Z 473.461,A -85,B 0,C 180,E1 -4278.975,E2 -4278.975} C_VEL
LIN {X 0,Y 530.95,Z 473.468,A -85,B 0,C 180,E1 -4281.529,E2 -4281.529} C_VEL
LIN {X 0,Y 530.974,Z 473.47,A -85,B 0,C 180,E1 -4284.382,E2 -4284.382} C_VEL
LIN {X 0,Y 530.966,Z 473.466,A -85,B 0,C 180,E1 -4287.134,E2 -4287.134} C_VEL
LIN {X 0,Y 530.976,Z 473.461,A -85,B 0,C 180,E1 -4289.804,E2 -4289.804} C_VEL
LIN {X 0,Y 531.008,Z 473.467,A -85,B 0,C 180,E1 -4292.466,E2 -4292.466} C_VEL
LIN {X 0,Y 530.998,Z 473.458,A -85,B 0,C 180,E1 -4294.943,E2 -4294.943} C_VEL
LIN {X 0,Y 530.961,Z 473.472,A -85,B 0,C 180,E1 -4298.247,E2 -4298.247} C_VEL
LIN {X 0,Y 530.987,Z 473.464,A -85,B 0,C 180,E1 -4300.677,E2 -4300.677} C_VEL
LIN {X 0,Y 530.983,Z 473.46,A -85,B 0,C 180,E1 -4303.071,E2 -4303.071} C_VEL
LIN {X 0,Y 531.008,Z 473.46,A -85,B 0,C 180,E1 -4305.436,E2 -4305.436} C_VEL
LIN {X 0,Y 531.036,Z 473.459,A -85,B 0,C 180,E1 -4308.55,E2 -4308.55} C_VEL
LIN {X 0,Y 531.05,Z 473.451,A -85,B 0,C 180,E1 -4311.63,E2 -4311.63} C_VEL
LIN {X 0,Y 531.131,Z 473.449,A -85,B 0,C 180,E1 -4314.686,E2 -4314.686} C_VEL
LIN {X 0,Y 531.13,Z 473.438,A -85,B 0,C 180,E1 -4317.725,E2 -4317.725} C_VEL
LIN {X 0,Y 531.146,Z 473.448,A -85,B 0,C 180,E1 -4320.759,E2 -4320.759} C_VEL
LIN {X 0,Y 531.1,Z 473.449,A -85,B 0,C 180,E1 -4323.035,E2 -4323.035} C_VEL
LIN {X 0,Y 531.075,Z 473.447,A -85,B 0,C 180,E1 -4326.078,E2 -4326.078} C_VEL
LIN {X 0,Y 531.027,Z 473.459,A -85,B 0,C 180,E1 -4329.139,E2 -4329.139} C_VEL
LIN {X 0,Y 531.032,Z 473.46,A -85,B 0,C 180,E1 -4332.225,E2 -4332.225} C_VEL
LIN {X 0,Y 530.987,Z 473.462,A -85,B 0,C 180,E1 -4335.35,E2 -4335.35} C_VEL
LIN {X 0,Y 531.008,Z 473.46,A -85,B 0,C 180,E1 -4337.723,E2 -4337.723} C_VEL
LIN {X 0,Y 530.994,Z 473.463,A -85,B 0,C 180,E1 -4340.938,E2 -4340.938} C_VEL
LIN {X 0,Y 530.973,Z 473.468,A -85,B 0,C 180,E1 -4344.225,E2 -4344.225} C_VEL
LIN {X 0,Y 531.005,Z 473.463,A -85,B 0,C 180,E1 -4346.744,E2 -4346.744} C_VEL
LIN {X 0,Y 530.976,Z 473.465,A -85,B 0,C 180,E1 -4349.323,E2 -4349.323} C_VEL
LIN {X 0,Y 530.974,Z 473.465,A -85,B 0,C 180,E1 -4352.104,E2 -4352.104} C_VEL
LIN {X 0,Y 530.984,Z 473.47,A -85,B 0,C 180,E1 -4354.855,E2 -4354.855} C_VEL
LIN {X 0,Y 530.961,Z 473.464,A -85,B 0,C 180,E1 -4357.508,E2 -4357.508} C_VEL
LIN {X 0,Y 530.996,Z 473.467,A -85,B 0,C 180,E1 -4360.432,E2 -4360.432} C_VEL
LIN {X 0,Y 530.95,Z 473.469,A -85,B 0,C 180,E1 -4363.496,E2 -4363.496} C_VEL
LIN {X 0,Y 530.963,Z 473.467,A -85,B 0,C 180,E1 -4366.506,E2 -4366.506} C_VEL
LIN {X 0,Y 530.987,Z 473.47,A -85,B 0,C 180,E1 -4368.976,E2 -4368.976} C_VEL
LIN {X 0,Y 530.956,Z 473.46,A -85,B 0,C 180,E1 -4371.53,E2 -4371.53} C_VEL
LIN {X 0,Y 530.953,Z 473.454,A -85,B 0,C 180,E1 -4374.381,E2 -4374.381} C_VEL
LIN {X 0,Y 530.967,Z 473.468,A -85,B 0,C 180,E1 -4377.134,E2 -4377.134} C_VEL
LIN {X 0,Y 530.969,Z 473.462,A -85,B 0,C 180,E1 -4379.804,E2 -4379.804} C_VEL
LIN {X 0,Y 531.043,Z 473.575,A -85,B 0,C 180,E1 -4382.697,E2 -4382.697} C_VEL
LIN {X 0,Y 532.611,Z 482.263,A -85,B 0,C 180,E1 -4384.397,E2 -4384.397} C_VEL
LIN {X 0,Y 532.214,Z 499.949,A -85,B 0,C 180,E1 -4387.484,E2 -4387.484} C_VEL
LIN {X 0,Y 531.81,Z 515.247,A -85,B 0,C 180,E1 -4390.106,E2 -4390.106} C_VEL
LIN {X 0,Y 531.629,Z 525.835,A -85,B 0,C 180,E1 -4391.868,E2 -4391.868} C_VEL
LIN {X 0,Y 533.875,Z 537.064,A -85,B 0,C 180,E1 -4392.125,E2 -4392.125} C_VEL
LIN {X 0,Y 533.283,Z 661.002,A -85,B 0,C 180,E1 -4393.836,E2 -4393.836} C_VEL
LIN {X 0,Y 533.137,Z 672.118,A -85,B 0,C 180,E1 -4394.081,E2 -4394.081} C_VEL
LIN {X 0,Y 532.959,Z 682.398,A -85,B 0,C 180,E1 -4394.395,E2 -4394.395} C_VEL
LIN {X 0,Y 532.724,Z 692.75,A -85,B 0,C 180,E1 -4394.8,E2 -4394.8} C_VEL
LIN {X 0,Y 532.483,Z 702.727,A -85,B 0,C 180,E1 -4395.282,E2 -4395.282} C_VEL
LIN {X 0,Y 532.214,Z 712.653,A -85,B 0,C 180,E1 -4395.86,E2 -4395.86} C_VEL
LIN {X 0,Y 531.95,Z 722.353,A -85,B 0,C 180,E1 -4396.535,E2 -4396.535} C_VEL
LIN {X 0,Y 531.675,Z 731.741,A -85,B 0,C 180,E1 -4397.305,E2 -4397.305} C_VEL
LIN {X 0,Y 531.393,Z 740.558,A -85,B 0,C 180,E1 -4398.153,E2 -4398.153} C_VEL
LIN {X 0,Y 531.235,Z 747.675,A -85,B 0,C 180,E1 -4398.941,E2 -4398.941} C_VEL
LIN {X 0,Y 530.987,Z 755.161,A -85,B 0,C 180,E1 -4399.9,E2 -4399.9} C_VEL
LIN {X 0,Y 530.822,Z 762.729,A -85,B 0,C 180,E1 -4401.05,E2 -4401.05} C_VEL
LIN {X 0,Y 530.698,Z 768.099,A -85,B 0,C 180,E1 -4402.007,E2 -4402.007} C_VEL
LIN {X 0,Y 530.573,Z 773.491,A -85,B 0,C 180,E1 -4403.153,E2 -4403.153} C_VEL
LIN {X 0,Y 530.563,Z 777.898,A -85,B 0,C 180,E1 -4404.299,E2 -4404.299} C_VEL
LIN {X 0,Y 530.448,Z 781.413,A -85,B 0,C 180,E1 -4405.441,E2 -4405.441} C_VEL
LIN {X 0,Y 530.497,Z 783.327,A -85,B 0,C 180,E1 -4406.202,E2 -4406.202} C_VEL
LIN {X 0,Y 530.408,Z 785.986,A -85,B 0,C 180,E1 -4407.722,E2 -4407.722} C_VEL
LIN {X 0,Y 530.341,Z 787.263,A -85,B 0,C 180,E1 -4409.241,E2 -4409.241} C_VEL
LIN {X 0,Y 530.341,Z 787.5,A -85,B 0,C 180,E1 -4410,E2 -4410} C_VEL
LIN {X 0,Y 530.356,Z 786.793,A -85,B 0,C 180,E1 -4411.519,E2 -4411.519} C_VEL
LIN {X 0,Y 530.408,Z 785.986,A -85,B 0,C 180,E1 -4412.278,E2 -4412.278} C_VEL
LIN {X 0,Y 530.497,Z 783.327,A -85,B 0,C 180,E1 -4413.798,E2 -4413.798} C_VEL
LIN {X 0,Y 530.513,Z 779.153,A -85,B 0,C 180,E1 -4415.321,E2 -4415.321} C_VEL
LIN {X 0,Y 530.573,Z 774.674,A -85,B 0,C 180,E1 -4416.558,E2 -4416.558} C_VEL
LIN {X 0,Y 530.641,Z 769.999,A -85,B 0,C 180,E1 -4417.611,E2 -4417.611} C_VEL
LIN {X 0,Y 530.768,Z 763.859,A -85,B 0,C 180,E1 -4418.758,E2 -4418.758} C_VEL
LIN {X 0,Y 530.92,Z 757.822,A -85,B 0,C 180,E1 -4419.716,E2 -4419.716} C_VEL
LIN {X 0,Y 531.152,Z 750.785,A -85,B 0,C 180,E1 -4420.675,E2 -4420.675} C_VEL
LIN {X 0,Y 531.344,Z 743.343,A -85,B 0,C 180,E1 -4421.551,E2 -4421.551} C_VEL
LIN {X 0,Y 531.576,Z 733.853,A -85,B 0,C 180,E1 -4422.503,E2 -4422.503} C_VEL
LIN {X 0,Y 531.853,Z 724.826,A -85,B 0,C 180,E1 -4423.273,E2 -4423.273} C_VEL
LIN {X 0,Y 532.083,Z 715.576,A -85,B 0,C 180,E1 -4423.948,E2 -4423.948} C_VEL
LIN {X 0,Y 532.422,Z 706.237,A -85,B 0,C 180,E1 -4424.525,E2 -4424.525} C_VEL
LIN {X 0,Y 532.681,Z 695.973,A -85,B 0,C 180,E1 -4425.055,E2 -4425.055} C_VEL
LIN {X 0,Y 532.927,Z 684.651,A -85,B 0,C 180,E1 -4425.525,E2 -4425.525} C_VEL
LIN {X 0,Y 533.067,Z 674.186,A -85,B 0,C 180,E1 -4425.865,E2 -4425.865} C_VEL
LIN {X 0,Y 533.251,Z 662.361,A -85,B 0,C 180,E1 -4426.141,E2 -4426.141} C_VEL
LIN {X 0,Y 533.464,Z 632.249,A -85,B 0,C 180,E1 -4426.577,E2 -4426.577} C_VEL
LIN {X 0,Y 533.868,Z 537.252,A -85,B 0,C 180,E1 -4427.873,E2 -4427.873} C_VEL
LIN {X 0,Y 531.638,Z 525.83,A -85,B 0,C 180,E1 -4428.132,E2 -4428.132} C_VEL
LIN {X 0,Y 532.009,Z 509.367,A -85,B 0,C 180,E1 -4430.896,E2 -4430.896} C_VEL
LIN {X 0,Y 532.366,Z 492.879,A -85,B 0,C 180,E1 -4433.743,E2 -4433.743} C_VEL
LIN {X 0,Y 532.596,Z 482.321,A -85,B 0,C 180,E1 -4435.604,E2 -4435.604} C_VEL
LIN {X 0,Y 531.043,Z 473.53,A -85,B 0,C 180,E1 -4437.303,E2 -4437.303} C_VEL
LIN {X 0,Y 530.969,Z 473.462,A -85,B 0,C 180,E1 -4440.196,E2 -4440.196} C_VEL
LIN {X 0,Y 530.967,Z 473.468,A -85,B 0,C 180,E1 -4442.866,E2 -4442.866} C_VEL
LIN {X 0,Y 530.953,Z 473.454,A -85,B 0,C 180,E1 -4445.619,E2 -4445.619} C_VEL
LIN {X 0,Y 530.966,Z 473.46,A -85,B 0,C 180,E1 -4448.653,E2 -4448.653} C_VEL
LIN {X 0,Y 530.997,Z 473.466,A -85,B 0,C 180,E1 -4451.434,E2 -4451.434} C_VEL
LIN {X 0,Y 530.984,Z 473.46,A -85,B 0,C 180,E1 -4454.546,E2 -4454.546} C_VEL
LIN {X 0,Y 530.979,Z 473.464,A -85,B 0,C 180,E1 -4457.833,E2 -4457.833} C_VEL
LIN {X 0,Y 530.985,Z 473.464,A -85,B 0,C 180,E1 -4460.556,E2 -4460.556} C_VEL
LIN {X 0,Y 530.968,Z 473.467,A -85,B 0,C 180,E1 -4463.842,E2 -4463.842} C_VEL
LIN {X 0,Y 530.993,Z 473.459,A -85,B 0,C 180,E1 -4466.493,E2 -4466.493} C_VEL
LIN {X 0,Y 530.968,Z 473.474,A -85,B 0,C 180,E1 -4469.354,E2 -4469.354} C_VEL
LIN {X 0,Y 531.011,Z 473.455,A -85,B 0,C 180,E1 -4472.466,E2 -4472.466} C_VEL
LIN {X 0,Y 531.001,Z 473.463,A -85,B 0,C 180,E1 -4474.942,E2 -4474.942} C_VEL
LIN {X 0,Y 530.964,Z 473.462,A -85,B 0,C 180,E1 -4478.246,E2 -4478.246} C_VEL
LIN {X 0,Y 530.989,Z 473.459,A -85,B 0,C 180,E1 -4480.677,E2 -4480.677} C_VEL
LIN {X 0,Y 530.985,Z 473.467,A -85,B 0,C 180,E1 -4483.071,E2 -4483.071} C_VEL
LIN {X 0,Y 531.01,Z 473.462,A -85,B 0,C 180,E1 -4485.435,E2 -4485.435} C_VEL
LIN {X 0,Y 531.027,Z 473.456,A -85,B 0,C 180,E1 -4488.549,E2 -4488.549} C_VEL
LIN {X 0,Y 531.051,Z 473.459,A -85,B 0,C 180,E1 -4491.629,E2 -4491.629} C_VEL
LIN {X 0,Y 531.115,Z 473.439,A -85,B 0,C 180,E1 -4494.685,E2 -4494.685} C_VEL
LIN {X 0,Y 531.131,Z 473.45,A -85,B 0,C 180,E1 -4497.725,E2 -4497.725} C_VEL
LIN {X 0,Y 531.146,Z 473.44,A -85,B 0,C 180,E1 -4500.758,E2 -4500.758} C_VEL
LIN {X 0,Y 531.1,Z 473.444,A -85,B 0,C 180,E1 -4503.034,E2 -4503.034} C_VEL
LIN {X 0,Y 531.074,Z 473.453,A -85,B 0,C 180,E1 -4506.077,E2 -4506.077} C_VEL
LIN {X 0,Y 531.026,Z 473.457,A -85,B 0,C 180,E1 -4509.138,E2 -4509.138} C_VEL
LIN {X 0,Y 531.031,Z 473.458,A -85,B 0,C 180,E1 -4512.225,E2 -4512.225} C_VEL
LIN {X 0,Y 530.986,Z 473.468,A -85,B 0,C 180,E1 -4515.35,E2 -4515.35} C_VEL
LIN {X 0,Y 531.006,Z 473.463,A -85,B 0,C 180,E1 -4517.722,E2 -4517.722} C_VEL
LIN {X 0,Y 530.992,Z 473.463,A -85,B 0,C 180,E1 -4520.938,E2 -4520.938} C_VEL
LIN {X 0,Y 530.97,Z 473.461,A -85,B 0,C 180,E1 -4524.224,E2 -4524.224} C_VEL
LIN {X 0,Y 531.002,Z 473.46,A -85,B 0,C 180,E1 -4526.743,E2 -4526.743} C_VEL
LIN {X 0,Y 530.991,Z 473.466,A -85,B 0,C 180,E1 -4529.322,E2 -4529.322} C_VEL
LIN {X 0,Y 530.971,Z 473.468,A -85,B 0,C 180,E1 -4532.103,E2 -4532.103} C_VEL
LIN {X 0,Y 530.982,Z 473.462,A -85,B 0,C 180,E1 -4534.855,E2 -4534.855} C_VEL
LIN {X 0,Y 530.957,Z 473.471,A -85,B 0,C 180,E1 -4537.508,E2 -4537.508} C_VEL
LIN {X 0,Y 530.976,Z 473.461,A -85,B 0,C 180,E1 -4540.433,E2 -4540.433} C_VEL
LIN {X 0,Y 530.961,Z 473.469,A -85,B 0,C 180,E1 -4543.282,E2 -4543.282} C_VEL
LIN {X 0,Y 530.954,Z 473.472,A -85,B 0,C 180,E1 -4543.578,E2 -4543.578} C_VEL
LIN {X 0,Y 530.281,Z 473.552,A -85,B 0,C 180,E1 -4544.212,E2 -4544.212} C_VEL
LIN {X 0,Y 527.434,Z 473.906,A -85,B 0,C 180,E1 -4545.241,E2 -4545.241} C_VEL
LIN {X 0,Y 525.031,Z 474.196,A -85,B 0,C 180,E1 -4546.069,E2 -4546.069} C_VEL
LIN {X 0,Y 524.001,Z 474.319,A -85,B 0,C 180,E1 -4546.709,E2 -4546.709} C_VEL
LIN {X 0,Y 523.917,Z 474.329,A -85,B 0,C 180,E1 -4546.925,E2 -4546.925} C_VEL
LIN {X 0,Y 523.971,Z 474.345,A -85,B 0,C 180,E1 -4549.924,E2 -4549.924} C_VEL
LIN {X 0,Y 523.905,Z 474.338,A -85,B 0,C 180,E1 -4552.869,E2 -4552.869} C_VEL
LIN {X 0,Y 523.937,Z 474.348,A -85,B 0,C 180,E1 -4555.711,E2 -4555.711} C_VEL
LIN {X 0,Y 523.927,Z 474.345,A -85,B 0,C 180,E1 -4558.457,E2 -4558.457} C_VEL
LIN {X 0,Y 523.945,Z 474.342,A -85,B 0,C 180,E1 -4561.126,E2 -4561.126} C_VEL
LIN {X 0,Y 523.979,Z 474.344,A -85,B 0,C 180,E1 -4563.98,E2 -4563.98} C_VEL
LIN {X 0,Y 523.931,Z 474.347,A -85,B 0,C 180,E1 -4566.271,E2 -4566.271} C_VEL
LIN {X 0,Y 523.941,Z 474.342,A -85,B 0,C 180,E1 -4568.767,E2 -4568.767} C_VEL
LIN {X 0,Y 523.949,Z 474.342,A -85,B 0,C 180,E1 -4571.221,E2 -4571.221} C_VEL
LIN {X 0,Y 523.934,Z 474.349,A -85,B 0,C 180,E1 -4573.639,E2 -4573.639} C_VEL
LIN {X 0,Y 523.937,Z 474.349,A -85,B 0,C 180,E1 -4576.028,E2 -4576.028} C_VEL
LIN {X 0,Y 524.008,Z 474.337,A -85,B 0,C 180,E1 -4578.394,E2 -4578.394} C_VEL
LIN {X 0,Y 524,Z 474.338,A -85,B 0,C 180,E1 -4581.516,E2 -4581.516} C_VEL
LIN {X 0,Y 524.078,Z 474.327,A -85,B 0,C 180,E1 -4584.614,E2 -4584.614} C_VEL
LIN {X 0,Y 524.11,Z 474.327,A -85,B 0,C 180,E1 -4587.695,E2 -4587.695} C_VEL
LIN {X 0,Y 524.119,Z 474.321,A -85,B 0,C 180,E1 -4590.768,E2 -4590.768} C_VEL
LIN {X 0,Y 524.069,Z 474.327,A -85,B 0,C 180,E1 -4593.075,E2 -4593.075} C_VEL
LIN {X 0,Y 524.043,Z 474.336,A -85,B 0,C 180,E1 -4596.159,E2 -4596.159} C_VEL
LIN {X 0,Y 523.994,Z 474.336,A -85,B 0,C 180,E1 -4599.262,E2 -4599.262} C_VEL
LIN {X 0,Y 523.999,Z 474.34,A -85,B 0,C 180,E1 -4601.739,E2 -4601.739} C_VEL
LIN {X 0,Y 523.989,Z 474.337,A -85,B 0,C 180,E1 -4605.052,E2 -4605.052} C_VEL
LIN {X 0,Y 523.96,Z 474.347,A -85,B 0,C 180,E1 -4607.969,E2 -4607.969} C_VEL
LIN {X 0,Y 523.967,Z 474.344,A -85,B 0,C 180,E1 -4610.41,E2 -4610.41} C_VEL
LIN {X 0,Y 523.912,Z 474.346,A -85,B 0,C 180,E1 -4612.893,E2 -4612.893} C_VEL
LIN {X 0,Y 523.947,Z 474.342,A -85,B 0,C 180,E1 -4615.418,E2 -4615.418} C_VEL
LIN {X 0,Y 523.965,Z 474.346,A -85,B 0,C 180,E1 -4617.998,E2 -4617.998} C_VEL
LIN {X 0,Y 523.947,Z 474.342,A -85,B 0,C 180,E1 -4620.856,E2 -4620.856} C_VEL
LIN {X 0,Y 523.955,Z 474.343,A -85,B 0,C 180,E1 -4623.735,E2 -4623.735} C_VEL
LIN {X 0,Y 523.915,Z 474.341,A -85,B 0,C 180,E1 -4626.404,E2 -4626.404} C_VEL
LIN {X 0,Y 523.953,Z 474.34,A -85,B 0,C 180,E1 -4629.081,E2 -4629.081} C_VEL
LIN {X 0,Y 523.951,Z 474.337,A -85,B 0,C 180,E1 -4632.118,E2 -4632.118} C_VEL
LIN {X 0,Y 523.948,Z 474.337,A -85,B 0,C 180,E1 -4635.308,E2 -4635.308} C_VEL
LIN {X 0,Y 523.953,Z 474.339,A -85,B 0,C 180,E1 -4638.689,E2 -4638.689} C_VEL
LIN {X 0,Y 523.908,Z 474.349,A -85,B 0,C 180,E1 -4641.898,E2 -4641.898} C_VEL
LIN {X 0,Y 523.931,Z 474.342,A -85,B 0,C 180,E1 -4644.908,E2 -4644.908} C_VEL
LIN {X 0,Y 523.934,Z 474.343,A -85,B 0,C 180,E1 -4647.678,E2 -4647.678} C_VEL
LIN {X 0,Y 523.96,Z 474.342,A -85,B 0,C 180,E1 -4650.673,E2 -4650.673} C_VEL
LIN {X 0,Y 523.968,Z 474.338,A -85,B 0,C 180,E1 -4653.729,E2 -4653.729} C_VEL
LIN {X 0,Y 523.926,Z 474.343,A -85,B 0,C 180,E1 -4656.271,E2 -4656.271} C_VEL
LIN {X 0,Y 523.937,Z 474.345,A -85,B 0,C 180,E1 -4658.767,E2 -4658.767} C_VEL
LIN {X 0,Y 523.944,Z 474.337,A -85,B 0,C 180,E1 -4661.221,E2 -4661.221} C_VEL
LIN {X 0,Y 523.93,Z 474.337,A -85,B 0,C 180,E1 -4663.639,E2 -4663.639} C_VEL
LIN {X 0,Y 523.93,Z 474.345,A -85,B 0,C 180,E1 -4666.028,E2 -4666.028} C_VEL
LIN {X 0,Y 524.001,Z 474.337,A -85,B 0,C 180,E1 -4668.394,E2 -4668.394} C_VEL
LIN {X 0,Y 523.998,Z 474.329,A -85,B 0,C 180,E1 -4671.516,E2 -4671.516} C_VEL
LIN {X 0,Y 524.089,Z 474.327,A -85,B 0,C 180,E1 -4674.614,E2 -4674.614} C_VEL
LIN {X 0,Y 524.103,Z 474.312,A -85,B 0,C 180,E1 -4677.695,E2 -4677.695} C_VEL
LIN {X 0,Y 524.116,Z 474.323,A -85,B 0,C 180,E1 -4680.769,E2 -4680.769} C_VEL
LIN {X 0,Y 524.067,Z 474.324,A -85,B 0,C 180,E1 -4683.075,E2 -4683.075} C_VEL
LIN {X 0,Y 524.037,Z 474.324,A -85,B 0,C 180,E1 -4686.159,E2 -4686.159} C_VEL
LIN {X 0,Y 523.994,Z 474.335,A -85,B 0,C 180,E1 -4689.262,E2 -4689.262} C_VEL
LIN {X 0,Y 523.993,Z 474.332,A -85,B 0,C 180,E1 -4691.74,E2 -4691.74} C_VEL
LIN {X 0,Y 523.984,Z 474.336,A -85,B 0,C 180,E1 -4695.053,E2 -4695.053} C_VEL
LIN {X 0,Y 523.956,Z 474.34,A -85,B 0,C 180,E1 -4697.97,E2 -4697.97} C_VEL
LIN {X 0,Y 523.964,Z 474.339,A -85,B 0,C 180,E1 -4700.411,E2 -4700.411} C_VEL
LIN {X 0,Y 523.909,Z 474.35,A -85,B 0,C 180,E1 -4702.894,E2 -4702.894} C_VEL
LIN {X 0,Y 523.947,Z 474.338,A -85,B 0,C 180,E1 -4705.419,E2 -4705.419} C_VEL
LIN {X 0,Y 523.964,Z 474.334,A -85,B 0,C 180,E1 -4708,E2 -4708} C_VEL
LIN {X 0,Y 523.94,Z 474.346,A -85,B 0,C 180,E1 -4710.856,E2 -4710.856} C_VEL
LIN {X 0,Y 523.955,Z 474.335,A -85,B 0,C 180,E1 -4713.736,E2 -4713.736} C_VEL
LIN {X 0,Y 523.917,Z 474.349,A -85,B 0,C 180,E1 -4716.405,E2 -4716.405} C_VEL
LIN {X 0,Y 523.918,Z 474.348,A -85,B 0,C 180,E1 -4719.085,E2 -4719.085} C_VEL
LIN {X 0,Y 523.965,Z 474.338,A -85,B 0,C 180,E1 -4721.313,E2 -4721.313} C_VEL
LIN {X 0,Y 523.95,Z 474.347,A -85,B 0,C 180,E1 -4724.692,E2 -4724.692} C_VEL
LIN {X 0,Y 523.954,Z 474.336,A -85,B 0,C 180,E1 -4727.883,E2 -4727.883} C_VEL
LIN {X 0,Y 523.92,Z 474.342,A -85,B 0,C 180,E1 -4730.916,E2 -4730.916} C_VEL
LIN {X 0,Y 523.897,Z 474.329,A -85,B 0,C 180,E1 -4733.826,E2 -4733.826} C_VEL
LIN {X 0,Y 523.941,Z 474.349,A -85,B 0,C 180,E1 -4736.636,E2 -4736.636} C_VEL
LIN {X 0,Y 523.956,Z 474.33,A -85,B 0,C 180,E1 -4739.356,E2 -4739.356} C_VEL
LIN {X 0,Y 524,Z 474.491,A -85,B 0,C 180,E1 -4742.508,E2 -4742.508} C_VEL
LIN {X 0,Y 525.656,Z 483.292,A -85,B 0,C 180,E1 -4744.246,E2 -4744.246} C_VEL
LIN {X 0,Y 525.335,Z 498.611,A -85,B 0,C 180,E1 -4746.965,E2 -4746.965} C_VEL
LIN {X 0,Y 524.863,Z 515.089,A -85,B 0,C 180,E1 -4749.831,E2 -4749.831} C_VEL
LIN {X 0,Y 524.663,Z 525.532,A -85,B 0,C 180,E1 -4751.612,E2 -4751.612} C_VEL
LIN {X 0,Y 526.496,Z 534.978,A -85,B 0,C 180,E1 -4751.839,E2 -4751.839} C_VEL
LIN {X 0,Y 527.137,Z 540.12,A -85,B 0,C 180,E1 -4751.934,E2 -4751.934} C_VEL
LIN {X 0,Y 526.459,Z 660.804,A -85,B 0,C 180,E1 -4753.62,E2 -4753.62} C_VEL
LIN {X 0,Y 526.308,Z 671.757,A -85,B 0,C 180,E1 -4753.864,E2 -4753.864} C_VEL
LIN {X 0,Y 526.104,Z 682.2,A -85,B 0,C 180,E1 -4754.186,E2 -4754.186} C_VEL
LIN {X 0,Y 525.863,Z 692.551,A -85,B 0,C 180,E1 -4754.596,E2 -4754.596} C_VEL
LIN {X 0,Y 525.598,Z 702.528,A -85,B 0,C 180,E1 -4755.085,E2 -4755.085} C_VEL
LIN {X 0,Y 525.296,Z 712.454,A -85,B 0,C 180,E1 -4755.67,E2 -4755.67} C_VEL
LIN {X 0,Y 524.99,Z 722.185,A -85,B 0,C 180,E1 -4756.353,E2 -4756.353} C_VEL
LIN {X 0,Y 524.699,Z 731.611,A -85,B 0,C 180,E1 -4757.134,E2 -4757.134} C_VEL
LIN {X 0,Y 524.439,Z 739.94,A -85,B 0,C 180,E1 -4757.937,E2 -4757.937} C_VEL
LIN {X 0,Y 524.239,Z 747.617,A -85,B 0,C 180,E1 -4758.791,E2 -4758.791} C_VEL
LIN {X 0,Y 523.937,Z 755.14,A -85,B 0,C 180,E1 -4759.762,E2 -4759.762} C_VEL
LIN {X 0,Y 523.817,Z 761.591,A -85,B 0,C 180,E1 -4760.735,E2 -4760.735} C_VEL
LIN {X 0,Y 523.646,Z 768.091,A -85,B 0,C 180,E1 -4761.899,E2 -4761.899} C_VEL
LIN {X 0,Y 523.495,Z 773.484,A -85,B 0,C 180,E1 -4763.06,E2 -4763.06} C_VEL
LIN {X 0,Y 523.477,Z 777.892,A -85,B 0,C 180,E1 -4764.221,E2 -4764.221} C_VEL
LIN {X 0,Y 523.352,Z 781.406,A -85,B 0,C 180,E1 -4765.379,E2 -4765.379} C_VEL
LIN {X 0,Y 523.419,Z 783.326,A -85,B 0,C 180,E1 -4766.151,E2 -4766.151} C_VEL
LIN {X 0,Y 523.332,Z 785.981,A -85,B 0,C 180,E1 -4767.691,E2 -4767.691} C_VEL
LIN {X 0,Y 523.247,Z 787.257,A -85,B 0,C 180,E1 -4769.23,E2 -4769.23} C_VEL
LIN {X 0,Y 523.245,Z 787.5,A -85,B 0,C 180,E1 -4770,E2 -4770} C_VEL
LIN {X 0,Y 523.27,Z 786.788,A -85,B 0,C 180,E1 -4771.539,E2 -4771.539} C_VEL
LIN {X 0,Y 523.332,Z 785.981,A -85,B 0,C 180,E1 -4772.309,E2 -4772.309} C_VEL
LIN {X 0,Y 523.419,Z 783.326,A -85,B 0,C 180,E1 -4773.849,E2 -4773.849} C_VEL
LIN {X 0,Y 523.448,Z 779.148,A -85,B 0,C 180,E1 -4775.393,E2 -4775.393} C_VEL
LIN {X 0,Y 523.486,Z 775.078,A -85,B 0,C 180,E1 -4776.546,E2 -4776.546} C_VEL
LIN {X 0,Y 523.572,Z 769.991,A -85,B 0,C 180,E1 -4777.714,E2 -4777.714} C_VEL
LIN {X 0,Y 523.73,Z 763.853,A -85,B 0,C 180,E1 -4778.877,E2 -4778.877} C_VEL
LIN {X 0,Y 523.885,Z 757.813,A -85,B 0,C 180,E1 -4779.848,E2 -4779.848} C_VEL
LIN {X 0,Y 524.122,Z 750.741,A -85,B 0,C 180,E1 -4780.82,E2 -4780.82} C_VEL
LIN {X 0,Y 524.298,Z 742.966,A -85,B 0,C 180,E1 -4781.74,E2 -4781.74} C_VEL
LIN {X 0,Y 524.591,Z 733.73,A -85,B 0,C 180,E1 -4782.672,E2 -4782.672} C_VEL
LIN {X 0,Y 524.915,Z 724.667,A -85,B 0,C 180,E1 -4783.452,E2 -4783.452} C_VEL
LIN {X 0,Y 525.164,Z 715.384,A -85,B 0,C 180,E1 -4784.136,E2 -4784.136} C_VEL
LIN {X 0,Y 525.501,Z 706.038,A -85,B 0,C 180,E1 -4784.72,E2 -4784.72} C_VEL
LIN {X 0,Y 525.798,Z 695.774,A -85,B 0,C 180,E1 -4785.257,E2 -4785.257} C_VEL
LIN {X 0,Y 526.06,Z 684.382,A -85,B 0,C 180,E1 -4785.736,E2 -4785.736} C_VEL
LIN {X 0,Y 526.233,Z 673.145,A -85,B 0,C 180,E1 -4786.1,E2 -4786.1} C_VEL
LIN {X 0,Y 526.428,Z 662.163,A -85,B 0,C 180,E1 -4786.356,E2 -4786.356} C_VEL
LIN {X 0,Y 526.68,Z 632.051,A -85,B 0,C 180,E1 -4786.797,E2 -4786.797} C_VEL
LIN {X 0,Y 527.05,Z 537.799,A -85,B 0,C 180,E1 -4788.102,E2 -4788.102} C_VEL
LIN {X 0,Y 524.686,Z 525.949,A -85,B 0,C 180,E1 -4788.363,E2 -4788.363} C_VEL
LIN {X 0,Y 524.626,Z 524.818,A -85,B 0,C 180,E1 -4788.48,E2 -4788.48} C_VEL
LIN {X 0,Y 525.092,Z 506.853,A -85,B 0,C 180,E1 -4791.596,E2 -4791.596} C_VEL
LIN {X 0,Y 525.536,Z 490.389,A -85,B 0,C 180,E1 -4794.491,E2 -4794.491} C_VEL
LIN {X 0,Y 525.653,Z 483.355,A -85,B 0,C 180,E1 -4795.755,E2 -4795.755} C_VEL
LIN {X 0,Y 524,Z 474.463,A -85,B 0,C 180,E1 -4797.492,E2 -4797.492} C_VEL
LIN {X 0,Y 523.956,Z 474.33,A -85,B 0,C 180,E1 -4800.644,E2 -4800.644} C_VEL
LIN {X 0,Y 523.958,Z 474.342,A -85,B 0,C 180,E1 -4803.734,E2 -4803.734} C_VEL
LIN {X 0,Y 523.9,Z 474.327,A -85,B 0,C 180,E1 -4806.4,E2 -4806.4} C_VEL
LIN {X 0,Y 523.92,Z 474.342,A -85,B 0,C 180,E1 -4809.084,E2 -4809.084} C_VEL
LIN {X 0,Y 523.954,Z 474.336,A -85,B 0,C 180,E1 -4812.117,E2 -4812.117} C_VEL
LIN {X 0,Y 523.95,Z 474.346,A -85,B 0,C 180,E1 -4815.308,E2 -4815.308} C_VEL
LIN {X 0,Y 523.965,Z 474.337,A -85,B 0,C 180,E1 -4818.687,E2 -4818.687} C_VEL
LIN {X 0,Y 523.915,Z 474.35,A -85,B 0,C 180,E1 -4821.079,E2 -4821.079} C_VEL
LIN {X 0,Y 523.923,Z 474.345,A -85,B 0,C 180,E1 -4823.827,E2 -4823.827} C_VEL
LIN {X 0,Y 523.937,Z 474.339,A -85,B 0,C 180,E1 -4826.635,E2 -4826.635} C_VEL
LIN {X 0,Y 523.95,Z 474.348,A -85,B 0,C 180,E1 -4829.355,E2 -4829.355} C_VEL
LIN {X 0,Y 523.973,Z 474.332,A -85,B 0,C 180,E1 -4832.28,E2 -4832.28} C_VEL
LIN {X 0,Y 523.948,Z 474.338,A -85,B 0,C 180,E1 -4834.581,E2 -4834.581} C_VEL
LIN {X 0,Y 523.909,Z 474.35,A -85,B 0,C 180,E1 -4837.106,E2 -4837.106} C_VEL
LIN {X 0,Y 523.971,Z 474.336,A -85,B 0,C 180,E1 -4839.865,E2 -4839.865} C_VEL
LIN {X 0,Y 523.963,Z 474.339,A -85,B 0,C 180,E1 -4842.837,E2 -4842.837} C_VEL
LIN {X 0,Y 523.967,Z 474.342,A -85,B 0,C 180,E1 -4845.235,E2 -4845.235} C_VEL
LIN {X 0,Y 524.003,Z 474.331,A -85,B 0,C 180,E1 -4848.394,E2 -4848.394} C_VEL
LIN {X 0,Y 523.998,Z 474.339,A -85,B 0,C 180,E1 -4851.516,E2 -4851.516} C_VEL
LIN {X 0,Y 524.076,Z 474.315,A -85,B 0,C 180,E1 -4854.613,E2 -4854.613} C_VEL
LIN {X 0,Y 524.103,Z 474.326,A -85,B 0,C 180,E1 -4857.694,E2 -4857.694} C_VEL
LIN {X 0,Y 524.116,Z 474.315,A -85,B 0,C 180,E1 -4860.768,E2 -4860.768} C_VEL
LIN {X 0,Y 524.067,Z 474.32,A -85,B 0,C 180,E1 -4863.075,E2 -4863.075} C_VEL
LIN {X 0,Y 524.036,Z 474.329,A -85,B 0,C 180,E1 -4866.159,E2 -4866.159} C_VEL
LIN {X 0,Y 523.994,Z 474.334,A -85,B 0,C 180,E1 -4869.262,E2 -4869.262} C_VEL
LIN {X 0,Y 523.998,Z 474.339,A -85,B 0,C 180,E1 -4871.743,E2 -4871.743} C_VEL
LIN {X 0,Y 523.982,Z 474.337,A -85,B 0,C 180,E1 -4875.052,E2 -4875.052} C_VEL
LIN {X 0,Y 523.954,Z 474.339,A -85,B 0,C 180,E1 -4877.969,E2 -4877.969} C_VEL
LIN {X 0,Y 523.962,Z 474.338,A -85,B 0,C 180,E1 -4880.41,E2 -4880.41} C_VEL
LIN {X 0,Y 523.907,Z 474.344,A -85,B 0,C 180,E1 -4882.893,E2 -4882.893} C_VEL
LIN {X 0,Y 523.945,Z 474.34,A -85,B 0,C 180,E1 -4885.419,E2 -4885.419} C_VEL
LIN {X 0,Y 523.961,Z 474.342,A -85,B 0,C 180,E1 -4887.999,E2 -4887.999} C_VEL
LIN {X 0,Y 523.943,Z 474.335,A -85,B 0,C 180,E1 -4890.856,E2 -4890.856} C_VEL
LIN {X 0,Y 523.953,Z 474.347,A -85,B 0,C 180,E1 -4893.735,E2 -4893.735} C_VEL
LIN {X 0,Y 523.913,Z 474.342,A -85,B 0,C 180,E1 -4896.405,E2 -4896.405} C_VEL
LIN {X 0,Y 523.915,Z 474.346,A -85,B 0,C 180,E1 -4899.085,E2 -4899.085} C_VEL
LIN {X 0,Y 523.949,Z 474.344,A -85,B 0,C 180,E1 -4902.119,E2 -4902.119} C_VEL
LIN {X 0,Y 523.948,Z 474.34,A -85,B 0,C 180,E1 -4905.309,E2 -4905.309} C_VEL
LIN {X 0,Y 523.917,Z 474.329,A -85,B 0,C 180,E1 -4906.925,E2 -4906.925} C_VEL
LIN {X 0,Y 523.254,Z 474.419,A -85,B 0,C 180,E1 -4907.567,E2 -4907.567} C_VEL
LIN {X 0,Y 520.418,Z 474.78,A -85,B 0,C 180,E1 -4908.609,E2 -4908.609} C_VEL
LIN {X 0,Y 518.019,Z 475.084,A -85,B 0,C 180,E1 -4909.448,E2 -4909.448} C_VEL
LIN {X 0,Y 516.988,Z 475.213,A -85,B 0,C 180,E1 -4910.096,E2 -4910.096} C_VEL
LIN {X 0,Y 516.903,Z 475.22,A -85,B 0,C 180,E1 -4910.315,E2 -4910.315} C_VEL
LIN {X 0,Y 516.878,Z 475.216,A -85,B 0,C 180,E1 -4913.342,E2 -4913.342} C_VEL
LIN {X 0,Y 516.905,Z 475.223,A -85,B 0,C 180,E1 -4916.121,E2 -4916.121} C_VEL
LIN {X 0,Y 516.888,Z 475.22,A -85,B 0,C 180,E1 -4918.935,E2 -4918.935} C_VEL
LIN {X 0,Y 516.919,Z 475.222,A -85,B 0,C 180,E1 -4921.586,E2 -4921.586} C_VEL
LIN {X 0,Y 516.926,Z 475.22,A -85,B 0,C 180,E1 -4924.211,E2 -4924.211} C_VEL
LIN {X 0,Y 516.867,Z 475.223,A -85,B 0,C 180,E1 -4926.777,E2 -4926.777} C_VEL
LIN {X 0,Y 516.934,Z 475.222,A -85,B 0,C 180,E1 -4929.732,E2 -4929.732} C_VEL
LIN {X 0,Y 516.925,Z 475.218,A -85,B 0,C 180,E1 -4932.596,E2 -4932.596} C_VEL
LIN {X 0,Y 516.938,Z 475.215,A -85,B 0,C 180,E1 -4935.03,E2 -4935.03} C_VEL
LIN {X 0,Y 516.961,Z 475.217,A -85,B 0,C 180,E1 -4938.234,E2 -4938.234} C_VEL
LIN {X 0,Y 516.965,Z 475.213,A -85,B 0,C 180,E1 -4941.4,E2 -4941.4} C_VEL
LIN {X 0,Y 517.006,Z 475.213,A -85,B 0,C 180,E1 -4943.757,E2 -4943.757} C_VEL
LIN {X 0,Y 517.082,Z 475.202,A -85,B 0,C 180,E1 -4947.663,E2 -4947.663} C_VEL
LIN {X 0,Y 517.09,Z 475.197,A -85,B 0,C 180,E1 -4950.779,E2 -4950.779} C_VEL
LIN {X 0,Y 517.01,Z 475.207,A -85,B 0,C 180,E1 -4953.117,E2 -4953.117} C_VEL
LIN {X 0,Y 517.007,Z 475.213,A -85,B 0,C 180,E1 -4956.243,E2 -4956.243} C_VEL
LIN {X 0,Y 516.949,Z 475.215,A -85,B 0,C 180,E1 -4959.389,E2 -4959.389} C_VEL
LIN {X 0,Y 516.948,Z 475.219,A -85,B 0,C 180,E1 -4961.807,E2 -4961.807} C_VEL
LIN {X 0,Y 516.94,Z 475.215,A -85,B 0,C 180,E1 -4965.146,E2 -4965.146} C_VEL
LIN {X 0,Y 516.922,Z 475.223,A -85,B 0,C 180,E1 -4968.222,E2 -4968.222} C_VEL
LIN {X 0,Y 516.908,Z 475.22,A -85,B 0,C 180,E1 -4970.701,E2 -4970.701} C_VEL
LIN {X 0,Y 516.906,Z 475.225,A -85,B 0,C 180,E1 -4974.072,E2 -4974.072} C_VEL
LIN {X 0,Y 516.921,Z 475.219,A -85,B 0,C 180,E1 -4976.657,E2 -4976.657} C_VEL
LIN {X 0,Y 516.919,Z 475.218,A -85,B 0,C 180,E1 -4979.526,E2 -4979.526} C_VEL
LIN {X 0,Y 516.894,Z 475.224,A -85,B 0,C 180,E1 -4982.544,E2 -4982.544} C_VEL
LIN {X 0,Y 516.876,Z 475.22,A -85,B 0,C 180,E1 -4985.332,E2 -4985.332} C_VEL
LIN {X 0,Y 516.875,Z 475.219,A -85,B 0,C 180,E1 -4987.943,E2 -4987.943} C_VEL
LIN {X 0,Y 516.897,Z 475.218,A -85,B 0,C 180,E1 -4990.739,E2 -4990.739} C_VEL
LIN {X 0,Y 516.875,Z 475.21,A -85,B 0,C 180,E1 -4993.903,E2 -4993.903} C_VEL
LIN {X 0,Y 516.874,Z 475.226,A -85,B 0,C 180,E1 -4996.107,E2 -4996.107} C_VEL
LIN {X 0,Y 516.909,Z 475.22,A -85,B 0,C 180,E1 -4998.398,E2 -4998.398} C_VEL
LIN {X 0,Y 516.874,Z 475.221,A -85,B 0,C 180,E1 -5001.284,E2 -5001.284} C_VEL
LIN {X 0,Y 516.882,Z 475.223,A -85,B 0,C 180,E1 -5004.221,E2 -5004.221} C_VEL
LIN {X 0,Y 516.889,Z 475.22,A -85,B 0,C 180,E1 -5007.053,E2 -5007.053} C_VEL
LIN {X 0,Y 516.892,Z 475.215,A -85,B 0,C 180,E1 -5009.797,E2 -5009.797} C_VEL
LIN {X 0,Y 516.92,Z 475.222,A -85,B 0,C 180,E1 -5012.467,E2 -5012.467} C_VEL
LIN {X 0,Y 516.902,Z 475.212,A -85,B 0,C 180,E1 -5015.072,E2 -5015.072} C_VEL
LIN {X 0,Y 516.877,Z 475.229,A -85,B 0,C 180,E1 -5018.462,E2 -5018.462} C_VEL
LIN {X 0,Y 516.895,Z 475.216,A -85,B 0,C 180,E1 -5020.955,E2 -5020.955} C_VEL
LIN {X 0,Y 516.907,Z 475.211,A -85,B 0,C 180,E1 -5023.41,E2 -5023.41} C_VEL
LIN {X 0,Y 516.885,Z 475.221,A -85,B 0,C 180,E1 -5025.834,E2 -5025.834} C_VEL
LIN {X 0,Y 516.947,Z 475.207,A -85,B 0,C 180,E1 -5029.028,E2 -5029.028} C_VEL
LIN {X 0,Y 516.969,Z 475.21,A -85,B 0,C 180,E1 -5032.187,E2 -5032.187} C_VEL
LIN {X 0,Y 517.05,Z 475.205,A -85,B 0,C 180,E1 -5034.541,E2 -5034.541} C_VEL
LIN {X 0,Y 517.075,Z 475.187,A -85,B 0,C 180,E1 -5037.663,E2 -5037.663} C_VEL
LIN {X 0,Y 517.086,Z 475.199,A -85,B 0,C 180,E1 -5040.779,E2 -5040.779} C_VEL
LIN {X 0,Y 517.008,Z 475.203,A -85,B 0,C 180,E1 -5043.117,E2 -5043.117} C_VEL
LIN {X 0,Y 517.001,Z 475.2,A -85,B 0,C 180,E1 -5046.244,E2 -5046.244} C_VEL
LIN {X 0,Y 516.947,Z 475.212,A -85,B 0,C 180,E1 -5049.39,E2 -5049.39} C_VEL
LIN {X 0,Y 516.943,Z 475.211,A -85,B 0,C 180,E1 -5051.808,E2 -5051.808} C_VEL
LIN {X 0,Y 516.935,Z 475.213,A -85,B 0,C 180,E1 -5055.147,E2 -5055.147} C_VEL
LIN {X 0,Y 516.918,Z 475.219,A -85,B 0,C 180,E1 -5058.223,E2 -5058.223} C_VEL
LIN {X 0,Y 516.905,Z 475.217,A -85,B 0,C 180,E1 -5060.702,E2 -5060.702} C_VEL
LIN {X 0,Y 516.904,Z 475.219,A -85,B 0,C 180,E1 -5064.073,E2 -5064.073} C_VEL
LIN {X 0,Y 516.922,Z 475.217,A -85,B 0,C 180,E1 -5066.658,E2 -5066.658} C_VEL
LIN {X 0,Y 516.905,Z 475.217,A -85,B 0,C 180,E1 -5069.525,E2 -5069.525} C_VEL
LIN {X 0,Y 516.894,Z 475.222,A -85,B 0,C 180,E1 -5072.545,E2 -5072.545} C_VEL
LIN {X 0,Y 516.877,Z 475.222,A -85,B 0,C 180,E1 -5075.333,E2 -5075.333} C_VEL
LIN {X 0,Y 516.876,Z 475.218,A -85,B 0,C 180,E1 -5077.944,E2 -5077.944} C_VEL
LIN {X 0,Y 516.898,Z 475.226,A -85,B 0,C 180,E1 -5080.741,E2 -5080.741} C_VEL
LIN {X 0,Y 516.878,Z 475.222,A -85,B 0,C 180,E1 -5083.904,E2 -5083.904} C_VEL
LIN {X 0,Y 516.879,Z 475.218,A -85,B 0,C 180,E1 -5086.108,E2 -5086.108} C_VEL
LIN {X 0,Y 516.914,Z 475.217,A -85,B 0,C 180,E1 -5088.399,E2 -5088.399} C_VEL
LIN {X 0,Y 516.88,Z 475.214,A -85,B 0,C 180,E1 -5091.285,E2 -5091.285} C_VEL
LIN {X 0,Y 516.869,Z 475.205,A -85,B 0,C 180,E1 -5094.22,E2 -5094.22} C_VEL
LIN {X 0,Y 516.895,Z 475.222,A -85,B 0,C 180,E1 -5097.054,E2 -5097.054} C_VEL
LIN {X 0,Y 516.892,Z 475.212,A -85,B 0,C 180,E1 -5099.797,E2 -5099.797} C_VEL
LIN {X 0,Y 516.969,Z 475.336,A -85,B 0,C 180,E1 -5102.284,E2 -5102.284} C_VEL
LIN {X 0,Y 518.793,Z 485.492,A -85,B 0,C 180,E1 -5104.311,E2 -5104.311} C_VEL
LIN {X 0,Y 518.295,Z 502.398,A -85,B 0,C 180,E1 -5107.341,E2 -5107.341} C_VEL
LIN {X 0,Y 517.85,Z 517.394,A -85,B 0,C 180,E1 -5109.984,E2 -5109.984} C_VEL
LIN {X 0,Y 517.655,Z 525.316,A -85,B 0,C 180,E1 -5111.354,E2 -5111.354} C_VEL
LIN {X 0,Y 519.613,Z 535.455,A -85,B 0,C 180,E1 -5111.6,E2 -5111.6} C_VEL
LIN {X 0,Y 520.4,Z 540.49,A -85,B 0,C 180,E1 -5111.7,E2 -5111.7} C_VEL
LIN {X 0,Y 519.647,Z 660.606,A -85,B 0,C 180,E1 -5113.399,E2 -5113.399} C_VEL
LIN {X 0,Y 519.506,Z 671.22,A -85,B 0,C 180,E1 -5113.638,E2 -5113.638} C_VEL
LIN {X 0,Y 519.245,Z 682.06,A -85,B 0,C 180,E1 -5113.974,E2 -5113.974} C_VEL
LIN {X 0,Y 519.002,Z 692.353,A -85,B 0,C 180,E1 -5114.388,E2 -5114.388} C_VEL
LIN {X 0,Y 518.714,Z 702.329,A -85,B 0,C 180,E1 -5114.882,E2 -5114.882} C_VEL
LIN {X 0,Y 518.39,Z 712.255,A -85,B 0,C 180,E1 -5115.475,E2 -5115.475} C_VEL
LIN {X 0,Y 518.041,Z 721.985,A -85,B 0,C 180,E1 -5116.166,E2 -5116.166} C_VEL
LIN {X 0,Y 517.713,Z 731.411,A -85,B 0,C 180,E1 -5116.957,E2 -5116.957} C_VEL
LIN {X 0,Y 517.416,Z 740.42,A -85,B 0,C 180,E1 -5117.845,E2 -5117.845} C_VEL
LIN {X 0,Y 517.204,Z 747.417,A -85,B 0,C 180,E1 -5118.637,E2 -5118.637} C_VEL
LIN {X 0,Y 516.918,Z 754.941,A -85,B 0,C 180,E1 -5119.622,E2 -5119.622} C_VEL
LIN {X 0,Y 516.774,Z 761.418,A -85,B 0,C 180,E1 -5120.608,E2 -5120.608} C_VEL
LIN {X 0,Y 516.579,Z 767.956,A -85,B 0,C 180,E1 -5121.787,E2 -5121.787} C_VEL
LIN {X 0,Y 516.403,Z 773.383,A -85,B 0,C 180,E1 -5122.965,E2 -5122.965} C_VEL
LIN {X 0,Y 516.394,Z 777.824,A -85,B 0,C 180,E1 -5124.142,E2 -5124.142} C_VEL
LIN {X 0,Y 516.263,Z 781.36,A -85,B 0,C 180,E1 -5125.315,E2 -5125.315} C_VEL
LIN {X 0,Y 516.324,Z 783.297,A -85,B 0,C 180,E1 -5126.098,E2 -5126.098} C_VEL
LIN {X 0,Y 516.258,Z 785.971,A -85,B 0,C 180,E1 -5127.659,E2 -5127.659} C_VEL
LIN {X 0,Y 516.157,Z 787.249,A -85,B 0,C 180,E1 -5129.22,E2 -5129.22} C_VEL
LIN {X 0,Y 516.152,Z 787.499,A -85,B 0,C 180,E1 -5130,E2 -5130} C_VEL
LIN {X 0,Y 516.188,Z 786.781,A -85,B 0,C 180,E1 -5131.56,E2 -5131.56} C_VEL
LIN {X 0,Y 516.258,Z 785.971,A -85,B 0,C 180,E1 -5132.341,E2 -5132.341} C_VEL
LIN {X 0,Y 516.324,Z 783.297,A -85,B 0,C 180,E1 -5133.902,E2 -5133.902} C_VEL
LIN {X 0,Y 516.381,Z 779.089,A -85,B 0,C 180,E1 -5135.467,E2 -5135.467} C_VEL
LIN {X 0,Y 516.412,Z 774.906,A -85,B 0,C 180,E1 -5136.656,E2 -5136.656} C_VEL
LIN {X 0,Y 516.505,Z 769.867,A -85,B 0,C 180,E1 -5137.82,E2 -5137.82} C_VEL
LIN {X 0,Y 516.669,Z 763.692,A -85,B 0,C 180,E1 -5138.999,E2 -5138.999} C_VEL
LIN {X 0,Y 516.828,Z 757.617,A -85,B 0,C 180,E1 -5139.984,E2 -5139.984} C_VEL
LIN {X 0,Y 517.105,Z 750.542,A -85,B 0,C 180,E1 -5140.969,E2 -5140.969} C_VEL
LIN {X 0,Y 517.281,Z 743.465,A -85,B 0,C 180,E1 -5141.826,E2 -5141.826} C_VEL
LIN {X 0,Y 517.628,Z 733.531,A -85,B 0,C 180,E1 -5142.846,E2 -5142.846} C_VEL
LIN {X 0,Y 517.977,Z 724.468,A -85,B 0,C 180,E1 -5143.635,E2 -5143.635} C_VEL
LIN {X 0,Y 518.255,Z 715.185,A -85,B 0,C 180,E1 -5144.328,E2 -5144.328} C_VEL
LIN {X 0,Y 518.591,Z 705.839,A -85,B 0,C 180,E1 -5144.921,E2 -5144.921} C_VEL
LIN {X 0,Y 518.891,Z 695.574,A -85,B 0,C 180,E1 -5145.465,E2 -5145.465} C_VEL
LIN {X 0,Y 519.191,Z 685.409,A -85,B 0,C 180,E1 -5145.904,E2 -5145.904} C_VEL
LIN {X 0,Y 519.394,Z 673.498,A -85,B 0,C 180,E1 -5146.303,E2 -5146.303} C_VEL
LIN {X 0,Y 519.629,Z 661.965,A -85,B 0,C 180,E1 -5146.576,E2 -5146.576} C_VEL
LIN {X 0,Y 519.894,Z 631.853,A -85,B 0,C 180,E1 -5147.022,E2 -5147.022} C_VEL
LIN {X 0,Y 520.292,Z 538.836,A -85,B 0,C 180,E1 -5148.328,E2 -5148.328} C_VEL
LIN {X 0,Y 517.661,Z 525.44,A -85,B 0,C 180,E1 -5148.636,E2 -5148.636} C_VEL
LIN {X 0,Y 518.139,Z 507.871,A -85,B 0,C 180,E1 -5151.691,E2 -5151.691} C_VEL
LIN {X 0,Y 518.581,Z 492.636,A -85,B 0,C 180,E1 -5154.403,E2 -5154.403} C_VEL
LIN {X 0,Y 518.683,Z 484.436,A -85,B 0,C 180,E1 -5155.902,E2 -5155.902} C_VEL
LIN {X 0,Y 516.969,Z 475.328,A -85,B 0,C 180,E1 -5157.716,E2 -5157.716} C_VEL
LIN {X 0,Y 516.892,Z 475.213,A -85,B 0,C 180,E1 -5160.203,E2 -5160.203} C_VEL
LIN {X 0,Y 516.895,Z 475.222,A -85,B 0,C 180,E1 -5162.946,E2 -5162.946} C_VEL
LIN {X 0,Y 516.869,Z 475.205,A -85,B 0,C 180,E1 -5165.78,E2 -5165.78} C_VEL
LIN {X 0,Y 516.88,Z 475.214,A -85,B 0,C 180,E1 -5168.715,E2 -5168.715} C_VEL
LIN {X 0,Y 516.913,Z 475.215,A -85,B 0,C 180,E1 -5171.774,E2 -5171.774} C_VEL
LIN {X 0,Y 516.919,Z 475.217,A -85,B 0,C 180,E1 -5175.009,E2 -5175.009} C_VEL
LIN {X 0,Y 516.916,Z 475.214,A -85,B 0,C 180,E1 -5178.397,E2 -5178.397} C_VEL
LIN {X 0,Y 516.878,Z 475.226,A -85,B 0,C 180,E1 -5181.284,E2 -5181.284} C_VEL
LIN {X 0,Y 516.885,Z 475.22,A -85,B 0,C 180,E1 -5184.221,E2 -5184.221} C_VEL
LIN {X 0,Y 516.891,Z 475.22,A -85,B 0,C 180,E1 -5187.052,E2 -5187.052} C_VEL
LIN {X 0,Y 516.886,Z 475.222,A -85,B 0,C 180,E1 -5189.796,E2 -5189.796} C_VEL
LIN {X 0,Y 516.923,Z 475.21,A -85,B 0,C 180,E1 -5192.467,E2 -5192.467} C_VEL
LIN {X 0,Y 516.904,Z 475.22,A -85,B 0,C 180,E1 -5195.071,E2 -5195.071} C_VEL
LIN {X 0,Y 516.879,Z 475.216,A -85,B 0,C 180,E1 -5198.462,E2 -5198.462} C_VEL
LIN {X 0,Y 516.897,Z 475.217,A -85,B 0,C 180,E1 -5200.954,E2 -5200.954} C_VEL
LIN {X 0,Y 516.909,Z 475.225,A -85,B 0,C 180,E1 -5203.41,E2 -5203.41} C_VEL
LIN {X 0,Y 516.886,Z 475.214,A -85,B 0,C 180,E1 -5205.833,E2 -5205.833} C_VEL
LIN {X 0,Y 516.956,Z 475.209,A -85,B 0,C 180,E1 -5208.233,E2 -5208.233} C_VEL
LIN {X 0,Y 516.963,Z 475.218,A -85,B 0,C 180,E1 -5211.399,E2 -5211.399} C_VEL
LIN {X 0,Y 517.001,Z 475.2,A -85,B 0,C 180,E1 -5213.756,E2 -5213.756} C_VEL
LIN {X 0,Y 517.075,Z 475.202,A -85,B 0,C 180,E1 -5217.663,E2 -5217.663} C_VEL
LIN {X 0,Y 517.086,Z 475.191,A -85,B 0,C 180,E1 -5220.778,E2 -5220.778} C_VEL
LIN {X 0,Y 517.008,Z 475.199,A -85,B 0,C 180,E1 -5223.117,E2 -5223.117} C_VEL
LIN {X 0,Y 517,Z 475.205,A -85,B 0,C 180,E1 -5226.243,E2 -5226.243} C_VEL
LIN {X 0,Y 516.948,Z 475.212,A -85,B 0,C 180,E1 -5229.389,E2 -5229.389} C_VEL
LIN {X 0,Y 516.947,Z 475.217,A -85,B 0,C 180,E1 -5231.81,E2 -5231.81} C_VEL
LIN {X 0,Y 516.933,Z 475.216,A -85,B 0,C 180,E1 -5235.146,E2 -5235.146} C_VEL
LIN {X 0,Y 516.916,Z 475.213,A -85,B 0,C 180,E1 -5238.222,E2 -5238.222} C_VEL
LIN {X 0,Y 516.903,Z 475.217,A -85,B 0,C 180,E1 -5240.701,E2 -5240.701} C_VEL
LIN {X 0,Y 516.901,Z 475.214,A -85,B 0,C 180,E1 -5244.072,E2 -5244.072} C_VEL
LIN {X 0,Y 516.919,Z 475.215,A -85,B 0,C 180,E1 -5246.658,E2 -5246.658} C_VEL
LIN {X 0,Y 516.915,Z 475.221,A -85,B 0,C 180,E1 -5249.527,E2 -5249.527} C_VEL
LIN {X 0,Y 516.892,Z 475.219,A -85,B 0,C 180,E1 -5252.545,E2 -5252.545} C_VEL
LIN {X 0,Y 516.875,Z 475.224,A -85,B 0,C 180,E1 -5255.333,E2 -5255.333} C_VEL
LIN {X 0,Y 516.873,Z 475.228,A -85,B 0,C 180,E1 -5257.944,E2 -5257.944} C_VEL
LIN {X 0,Y 516.877,Z 475.217,A -85,B 0,C 180,E1 -5260.742,E2 -5260.742} C_VEL
LIN {X 0,Y 516.896,Z 475.219,A -85,B 0,C 180,E1 -5262.829,E2 -5262.829} C_VEL
LIN {X 0,Y 516.914,Z 475.214,A -85,B 0,C 180,E1 -5265.01,E2 -5265.01} C_VEL
LIN {X 0,Y 516.922,Z 475.214,A -85,B 0,C 180,E1 -5268.397,E2 -5268.397} C_VEL
LIN {X 0,Y 516.903,Z 475.22,A -85,B 0,C 180,E1 -5270.315,E2 -5270.315} C_VEL
LIN {X 0,Y 516.234,Z 475.303,A -85,B 0,C 180,E1 -5270.965,E2 -5270.965} C_VEL
LIN {X 0,Y 513.377,Z 475.655,A -85,B 0,C 180,E1 -5272.021,E2 -5272.021} C_VEL
LIN {X 0,Y 510.957,Z 475.955,A -85,B 0,C 180,E1 -5272.871,E2 -5272.871} C_VEL
LIN {X 0,Y 509.912,Z 476.084,A -85,B 0,C 180,E1 -5273.527,E2 -5273.527} C_VEL
LIN {X 0,Y 509.824,Z 476.095,A -85,B 0,C 180,E1 -5273.749,E2 -5273.749} C_VEL
LIN {X 0,Y 509.856,Z 476.097,A -85,B 0,C 180,E1 -5276.54,E2 -5276.54} C_VEL
LIN {X 0,Y 509.845,Z 476.1,A -85,B 0,C 180,E1 -5279.335,E2 -5279.335} C_VEL
LIN {X 0,Y 509.889,Z 476.098,A -85,B 0,C 180,E1 -5282.055,E2 -5282.055} C_VEL
LIN {X 0,Y 509.872,Z 476.095,A -85,B 0,C 180,E1 -5284.704,E2 -5284.704} C_VEL
LIN {X 0,Y 509.831,Z 476.103,A -85,B 0,C 180,E1 -5287.455,E2 -5287.455} C_VEL
LIN {X 0,Y 509.912,Z 476.097,A -85,B 0,C 180,E1 -5289.845,E2 -5289.845} C_VEL
LIN {X 0,Y 509.88,Z 476.095,A -85,B 0,C 180,E1 -5293.175,E2 -5293.175} C_VEL
LIN {X 0,Y 509.86,Z 476.102,A -85,B 0,C 180,E1 -5295.634,E2 -5295.634} C_VEL
LIN {X 0,Y 509.909,Z 476.091,A -85,B 0,C 180,E1 -5298.875,E2 -5298.875} C_VEL
LIN {X 0,Y 509.948,Z 476.092,A -85,B 0,C 180,E1 -5302.079,E2 -5302.079} C_VEL
LIN {X 0,Y 509.977,Z 476.085,A -85,B 0,C 180,E1 -5304.464,E2 -5304.464} C_VEL
LIN {X 0,Y 510.053,Z 476.078,A -85,B 0,C 180,E1 -5307.631,E2 -5307.631} C_VEL
LIN {X 0,Y 510.06,Z 476.073,A -85,B 0,C 180,E1 -5310.789,E2 -5310.789} C_VEL
LIN {X 0,Y 509.952,Z 476.086,A -85,B 0,C 180,E1 -5313.16,E2 -5313.16} C_VEL
LIN {X 0,Y 509.975,Z 476.088,A -85,B 0,C 180,E1 -5316.329,E2 -5316.329} C_VEL
LIN {X 0,Y 509.911,Z 476.091,A -85,B 0,C 180,E1 -5318.72,E2 -5318.72} C_VEL
LIN {X 0,Y 509.9,Z 476.098,A -85,B 0,C 180,E1 -5321.931,E2 -5321.931} C_VEL
LIN {X 0,Y 509.889,Z 476.094,A -85,B 0,C 180,E1 -5325.242,E2 -5325.242} C_VEL
LIN {X 0,Y 509.884,Z 476.1,A -85,B 0,C 180,E1 -5328.001,E2 -5328.001} C_VEL
LIN {X 0,Y 509.845,Z 476.098,A -85,B 0,C 180,E1 -5331.001,E2 -5331.001} C_VEL
LIN {X 0,Y 509.832,Z 476.102,A -85,B 0,C 180,E1 -5333.563,E2 -5333.563} C_VEL
LIN {X 0,Y 509.906,Z 476.096,A -85,B 0,C 180,E1 -5336.378,E2 -5336.378} C_VEL
LIN {X 0,Y 509.88,Z 476.095,A -85,B 0,C 180,E1 -5338.843,E2 -5338.843} C_VEL
LIN {X 0,Y 509.82,Z 476.103,A -85,B 0,C 180,E1 -5341.589,E2 -5341.589} C_VEL
LIN {X 0,Y 509.847,Z 476.101,A -85,B 0,C 180,E1 -5344.413,E2 -5344.413} C_VEL
LIN {X 0,Y 509.812,Z 476.093,A -85,B 0,C 180,E1 -5347.34,E2 -5347.34} C_VEL
LIN {X 0,Y 509.854,Z 476.1,A -85,B 0,C 180,E1 -5350.38,E2 -5350.38} C_VEL
LIN {X 0,Y 509.832,Z 476.081,A -85,B 0,C 180,E1 -5353.064,E2 -5353.064} C_VEL
LIN {X 0,Y 509.822,Z 476.1,A -85,B 0,C 180,E1 -5355.792,E2 -5355.792} C_VEL
LIN {X 0,Y 509.85,Z 476.096,A -85,B 0,C 180,E1 -5358.575,E2 -5358.575} C_VEL
LIN {X 0,Y 509.843,Z 476.1,A -85,B 0,C 180,E1 -5361.786,E2 -5361.786} C_VEL
LIN {X 0,Y 509.838,Z 476.101,A -85,B 0,C 180,E1 -5364.623,E2 -5364.623} C_VEL
LIN {X 0,Y 509.857,Z 476.095,A -85,B 0,C 180,E1 -5367.481,E2 -5367.481} C_VEL
LIN {X 0,Y 509.872,Z 476.094,A -85,B 0,C 180,E1 -5370.269,E2 -5370.269} C_VEL
LIN {X 0,Y 509.878,Z 476.094,A -85,B 0,C 180,E1 -5372.944,E2 -5372.944} C_VEL
LIN {X 0,Y 509.86,Z 476.088,A -85,B 0,C 180,E1 -5375.574,E2 -5375.574} C_VEL
LIN {X 0,Y 509.841,Z 476.098,A -85,B 0,C 180,E1 -5378.998,E2 -5378.998} C_VEL
LIN {X 0,Y 509.878,Z 476.092,A -85,B 0,C 180,E1 -5381.999,E2 -5381.999} C_VEL
LIN {X 0,Y 509.9,Z 476.093,A -85,B 0,C 180,E1 -5384.819,E2 -5384.819} C_VEL
LIN {X 0,Y 509.895,Z 476.094,A -85,B 0,C 180,E1 -5388.121,E2 -5388.121} C_VEL
LIN {X 0,Y 509.909,Z 476.084,A -85,B 0,C 180,E1 -5391.28,E2 -5391.28} C_VEL
LIN {X 0,Y 509.969,Z 476.081,A -85,B 0,C 180,E1 -5393.671,E2 -5393.671} C_VEL
LIN {X 0,Y 509.95,Z 476.078,A -85,B 0,C 180,E1 -5396.84,E2 -5396.84} C_VEL
LIN {X 0,Y 510.056,Z 476.066,A -85,B 0,C 180,E1 -5399.211,E2 -5399.211} C_VEL
LIN {X 0,Y 510.046,Z 476.078,A -85,B 0,C 180,E1 -5402.369,E2 -5402.369} C_VEL
LIN {X 0,Y 509.969,Z 476.076,A -85,B 0,C 180,E1 -5406.33,E2 -5406.33} C_VEL
LIN {X 0,Y 509.909,Z 476.095,A -85,B 0,C 180,E1 -5408.721,E2 -5408.721} C_VEL
LIN {X 0,Y 509.895,Z 476.089,A -85,B 0,C 180,E1 -5411.932,E2 -5411.932} C_VEL
LIN {X 0,Y 509.885,Z 476.091,A -85,B 0,C 180,E1 -5415.242,E2 -5415.242} C_VEL
LIN {X 0,Y 509.88,Z 476.094,A -85,B 0,C 180,E1 -5418.002,E2 -5418.002} C_VEL
LIN {X 0,Y 509.843,Z 476.096,A -85,B 0,C 180,E1 -5421.002,E2 -5421.002} C_VEL
LIN {X 0,Y 509.829,Z 476.098,A -85,B 0,C 180,E1 -5423.564,E2 -5423.564} C_VEL
LIN {X 0,Y 509.906,Z 476.092,A -85,B 0,C 180,E1 -5426.38,E2 -5426.38} C_VEL
LIN {X 0,Y 509.871,Z 476.1,A -85,B 0,C 180,E1 -5428.845,E2 -5428.845} C_VEL
LIN {X 0,Y 509.819,Z 476.098,A -85,B 0,C 180,E1 -5431.591,E2 -5431.591} C_VEL
LIN {X 0,Y 509.848,Z 476.098,A -85,B 0,C 180,E1 -5434.414,E2 -5434.414} C_VEL
LIN {X 0,Y 509.814,Z 476.098,A -85,B 0,C 180,E1 -5437.341,E2 -5437.341} C_VEL
LIN {X 0,Y 509.855,Z 476.101,A -85,B 0,C 180,E1 -5440.381,E2 -5440.381} C_VEL
LIN {X 0,Y 509.818,Z 476.106,A -85,B 0,C 180,E1 -5443.063,E2 -5443.063} C_VEL
LIN {X 0,Y 509.827,Z 476.095,A -85,B 0,C 180,E1 -5445.793,E2 -5445.793} C_VEL
LIN {X 0,Y 509.856,Z 476.099,A -85,B 0,C 180,E1 -5448.576,E2 -5448.576} C_VEL
LIN {X 0,Y 509.849,Z 476.087,A -85,B 0,C 180,E1 -5451.787,E2 -5451.787} C_VEL
LIN {X 0,Y 509.829,Z 476.085,A -85,B 0,C 180,E1 -5454.623,E2 -5454.623} C_VEL
LIN {X 0,Y 509.863,Z 476.094,A -85,B 0,C 180,E1 -5457.482,E2 -5457.482} C_VEL
LIN {X 0,Y 509.858,Z 476.096,A -85,B 0,C 180,E1 -5460.274,E2 -5460.274} C_VEL
LIN {X 0,Y 509.893,Z 476.196,A -85,B 0,C 180,E1 -5462.055,E2 -5462.055} C_VEL
LIN {X 0,Y 511.839,Z 486.524,A -85,B 0,C 180,E1 -5464.155,E2 -5464.155} C_VEL
LIN {X 0,Y 511.399,Z 502.349,A -85,B 0,C 180,E1 -5467.038,E2 -5467.038} C_VEL
LIN {X 0,Y 510.853,Z 518.233,A -85,B 0,C 180,E1 -5469.884,E2 -5469.884} C_VEL
LIN {X 0,Y 510.686,Z 525.123,A -85,B 0,C 180,E1 -5471.092,E2 -5471.092} C_VEL
LIN {X 0,Y 513.293,Z 538.432,A -85,B 0,C 180,E1 -5471.41,E2 -5471.41} C_VEL
LIN {X 0,Y 513.655,Z 541.44,A -85,B 0,C 180,E1 -5471.467,E2 -5471.467} C_VEL
LIN {X 0,Y 512.851,Z 660.408,A -85,B 0,C 180,E1 -5473.173,E2 -5473.173} C_VEL
LIN {X 0,Y 512.692,Z 671.044,A -85,B 0,C 180,E1 -5473.415,E2 -5473.415} C_VEL
LIN {X 0,Y 512.415,Z 681.93,A -85,B 0,C 180,E1 -5473.757,E2 -5473.757} C_VEL
LIN {X 0,Y 512.157,Z 692.154,A -85,B 0,C 180,E1 -5474.173,E2 -5474.173} C_VEL
LIN {X 0,Y 511.843,Z 702.131,A -85,B 0,C 180,E1 -5474.674,E2 -5474.674} C_VEL
LIN {X 0,Y 511.496,Z 712.057,A -85,B 0,C 180,E1 -5475.275,E2 -5475.275} C_VEL
LIN {X 0,Y 511.079,Z 721.785,A -85,B 0,C 180,E1 -5475.974,E2 -5475.974} C_VEL
LIN {X 0,Y 510.738,Z 731.211,A -85,B 0,C 180,E1 -5476.776,E2 -5476.776} C_VEL
LIN {X 0,Y 510.411,Z 740.241,A -85,B 0,C 180,E1 -5477.678,E2 -5477.678} C_VEL
LIN {X 0,Y 510.176,Z 747.217,A -85,B 0,C 180,E1 -5478.478,E2 -5478.478} C_VEL
LIN {X 0,Y 509.9,Z 754.742,A -85,B 0,C 180,E1 -5479.477,E2 -5479.477} C_VEL
LIN {X 0,Y 509.675,Z 762.356,A -85,B 0,C 180,E1 -5480.676,E2 -5480.676} C_VEL
LIN {X 0,Y 509.497,Z 767.756,A -85,B 0,C 180,E1 -5481.672,E2 -5481.672} C_VEL
LIN {X 0,Y 509.328,Z 773.184,A -85,B 0,C 180,E1 -5482.866,E2 -5482.866} C_VEL
LIN {X 0,Y 509.291,Z 777.625,A -85,B 0,C 180,E1 -5484.06,E2 -5484.06} C_VEL
LIN {X 0,Y 509.18,Z 781.161,A -85,B 0,C 180,E1 -5485.25,E2 -5485.25} C_VEL
LIN {X 0,Y 509.217,Z 783.099,A -85,B 0,C 180,E1 -5486.043,E2 -5486.043} C_VEL
LIN {X 0,Y 509.187,Z 785.774,A -85,B 0,C 180,E1 -5487.627,E2 -5487.627} C_VEL
LIN {X 0,Y 509.071,Z 787.056,A -85,B 0,C 180,E1 -5489.209,E2 -5489.209} C_VEL
LIN {X 0,Y 509.064,Z 787.307,A -85,B 0,C 180,E1 -5490,E2 -5490} C_VEL
LIN {X 0,Y 509.109,Z 786.586,A -85,B 0,C 180,E1 -5491.582,E2 -5491.582} C_VEL
LIN {X 0,Y 509.187,Z 785.774,A -85,B 0,C 180,E1 -5492.373,E2 -5492.373} C_VEL
LIN {X 0,Y 509.217,Z 783.099,A -85,B 0,C 180,E1 -5493.957,E2 -5493.957} C_VEL
